// IOs for EL3446
	{attribute 'TcLinkTo' := 'TIID^Device 2 (EtherCAT)^Term 1 (EK1200)^Term 3 (EL3446)^I1 Channel^Overcurrent'}
	MDP5001_342_I1_Channel_Overcurrent_1						AT%I*  : BOOL;
	{attribute 'TcLinkTo' := 'TIID^Device 2 (EtherCAT)^Term 1 (EK1200)^Term 3 (EL3446)^I1 Channel^Inaccurate Current'}
	MDP5001_342_I1_Channel_Inaccurate_Current_1				AT%I*  : BOOL;
	{attribute 'TcLinkTo' := 'TIID^Device 2 (EtherCAT)^Term 1 (EK1200)^Term 3 (EL3446)^I1 Channel^Current Guard Warning'}
	MDP5001_342_I1_Channel_Current_Guard_Warning_1			AT%I*  : bool;
	{attribute 'TcLinkTo' := 'TIID^Device 2 (EtherCAT)^Term 1 (EK1200)^Term 3 (EL3446)^I1 Channel^Current Guard Error'}
	MDP5001_342_I1_Channel_Current_Guard_Error_1				AT%I*  : bool;
	{attribute 'TcLinkTo' := 'TIID^Device 2 (EtherCAT)^Term 1 (EK1200)^Term 3 (EL3446)^I1 Channel^Apparent Power Guard Warning'}
	MDP5001_342_I1_Channel_Apparent_Power_Guard_Warning_1		AT%I*  : bool;
	{attribute 'TcLinkTo' := 'TIID^Device 2 (EtherCAT)^Term 1 (EK1200)^Term 3 (EL3446)^I1 Channel^Apparent Power Guard Error'}
	MDP5001_342_I1_Channel_Apparent_Power_Guard_Error_1		AT%I*  : bool;
	{attribute 'TcLinkTo' := 'TIID^Device 2 (EtherCAT)^Term 1 (EK1200)^Term 3 (EL3446)^I1 Channel^Active Power Guard Warning'}
	MDP5001_342_I1_Channel_Active_Power_Guard_Warning_1		AT%I*  : bool;
	{attribute 'TcLinkTo' := 'TIID^Device 2 (EtherCAT)^Term 1 (EK1200)^Term 3 (EL3446)^I1 Channel^Active Power Guard Error'}
	MDP5001_342_I1_Channel_Active_Power_Guard_Error_1			AT%I*  : bool;
	{attribute 'TcLinkTo' := 'TIID^Device 2 (EtherCAT)^Term 1 (EK1200)^Term 3 (EL3446)^I1 Channel^Reactive Power Guard Warning'}
	MDP5001_342_I1_Channel_Reactive_Power_Guard_Warning_1		AT%I*  : bool;
	{attribute 'TcLinkTo' := 'TIID^Device 2 (EtherCAT)^Term 1 (EK1200)^Term 3 (EL3446)^I1 Channel^Reactive Power Guard Error'}
	MDP5001_342_I1_Channel_Reactive_Power_Guard_Error_1		AT%I*  : bool;
	{attribute 'TcLinkTo' := 'TIID^Device 2 (EtherCAT)^Term 1 (EK1200)^Term 3 (EL3446)^I1 Channel^DPM Inaccurate'}
	MDP5001_342_I1_Channel_DPM_Inaccurate_1					AT%I*  : bool;
	{attribute 'TcLinkTo' := 'TIID^Device 2 (EtherCAT)^Term 1 (EK1200)^Term 3 (EL3446)^I1 Channel^DPM Timeout'}
	MDP5001_342_I1_Channel_DPM_Timeout_1						AT%I*  : bool;
	{attribute 'TcLinkTo' := 'TIID^Device 2 (EtherCAT)^Term 1 (EK1200)^Term 3 (EL3446)^I1 Channel^TxPDO Toggle'}
	MDP5001_342_I1_Channel_TxPDO_Toggle_1						AT%I*  : bool;
	{attribute 'TcLinkTo' := 'TIID^Device 2 (EtherCAT)^Term 1 (EK1200)^Term 3 (EL3446)^I1 Channel^Current'}
	MDP5001_342_I1_Channel_Current_1							AT%I*  : REAL;
	{attribute 'TcLinkTo' := 'TIID^Device 2 (EtherCAT)^Term 1 (EK1200)^Term 3 (EL3446)^I1 Channel^Active Power'}
	MDP5001_342_I1_Channel_Active_Power_1						AT%I*  : REAL;
	{attribute 'TcLinkTo' := 'TIID^Device 2 (EtherCAT)^Term 1 (EK1200)^Term 3 (EL3446)^I1 Channel^Apparent Power'}
	MDP5001_342_I1_Channel_Apparent_Power_1					AT%I*  : REAL;
	{attribute 'TcLinkTo' := 'TIID^Device 2 (EtherCAT)^Term 1 (EK1200)^Term 3 (EL3446)^I1 Channel^Reactive Power Fundamental'}
	MDP5001_342_I1_Channel_Reactive_Power_Fundamental_1		AT%I*  : REAL;
	{attribute 'TcLinkTo' := 'TIID^Device 2 (EtherCAT)^Term 1 (EK1200)^Term 3 (EL3446)^I1 Channel^Active Energy'}
	MDP5001_342_I1_Channel_Active_Energy_1					AT%I*  : DINT;
	{attribute 'TcLinkTo' := 'TIID^Device 2 (EtherCAT)^Term 1 (EK1200)^Term 3 (EL3446)^I2 Channel^Overcurrent'}
	MDP5001_342_I2_Channel_Overcurrent_1						AT%I*  : BOOL;
	{attribute 'TcLinkTo' := 'TIID^Device 2 (EtherCAT)^Term 1 (EK1200)^Term 3 (EL3446)^I2 Channel^Inaccurate Current'}
	MDP5001_342_I2_Channel_Inaccurate_Current_1				AT%I*  : BOOL;
	{attribute 'TcLinkTo' := 'TIID^Device 2 (EtherCAT)^Term 1 (EK1200)^Term 3 (EL3446)^I2 Channel^Current Guard Warning'}
	MDP5001_342_I2_Channel_Current_Guard_Warning_1			AT%I*  : bool;
	{attribute 'TcLinkTo' := 'TIID^Device 2 (EtherCAT)^Term 1 (EK1200)^Term 3 (EL3446)^I2 Channel^Current Guard Error'}
	MDP5001_342_I2_Channel_Current_Guard_Error_1				AT%I*  : bool;
	{attribute 'TcLinkTo' := 'TIID^Device 2 (EtherCAT)^Term 1 (EK1200)^Term 3 (EL3446)^I2 Channel^Apparent Power Guard Warning'}
	MDP5001_342_I2_Channel_Apparent_Power_Guard_Warning_1		AT%I*  : bool;
	{attribute 'TcLinkTo' := 'TIID^Device 2 (EtherCAT)^Term 1 (EK1200)^Term 3 (EL3446)^I2 Channel^Apparent Power Guard Error'}
	MDP5001_342_I2_Channel_Apparent_Power_Guard_Error_1		AT%I*  : bool;
	{attribute 'TcLinkTo' := 'TIID^Device 2 (EtherCAT)^Term 1 (EK1200)^Term 3 (EL3446)^I2 Channel^Active Power Guard Warning'}
	MDP5001_342_I2_Channel_Active_Power_Guard_Warning_1		AT%I*  : bool;
	{attribute 'TcLinkTo' := 'TIID^Device 2 (EtherCAT)^Term 1 (EK1200)^Term 3 (EL3446)^I2 Channel^Active Power Guard Error'}
	MDP5001_342_I2_Channel_Active_Power_Guard_Error_1			AT%I*  : bool;
	{attribute 'TcLinkTo' := 'TIID^Device 2 (EtherCAT)^Term 1 (EK1200)^Term 3 (EL3446)^I2 Channel^Reactive Power Guard Warning'}
	MDP5001_342_I2_Channel_Reactive_Power_Guard_Warning_1		AT%I*  : bool;
	{attribute 'TcLinkTo' := 'TIID^Device 2 (EtherCAT)^Term 1 (EK1200)^Term 3 (EL3446)^I2 Channel^Reactive Power Guard Error'}
	MDP5001_342_I2_Channel_Reactive_Power_Guard_Error_1		AT%I*  : bool;
	{attribute 'TcLinkTo' := 'TIID^Device 2 (EtherCAT)^Term 1 (EK1200)^Term 3 (EL3446)^I2 Channel^DPM Inaccurate'}
	MDP5001_342_I2_Channel_DPM_Inaccurate_1					AT%I*  : bool;
	{attribute 'TcLinkTo' := 'TIID^Device 2 (EtherCAT)^Term 1 (EK1200)^Term 3 (EL3446)^I2 Channel^DPM Timeout'}
	MDP5001_342_I2_Channel_DPM_Timeout_1						AT%I*  : bool;
	{attribute 'TcLinkTo' := 'TIID^Device 2 (EtherCAT)^Term 1 (EK1200)^Term 3 (EL3446)^I2 Channel^TxPDO Toggle'}
	MDP5001_342_I2_Channel_TxPDO_Toggle_1						AT%I*  : bool;
	{attribute 'TcLinkTo' := 'TIID^Device 2 (EtherCAT)^Term 1 (EK1200)^Term 3 (EL3446)^I2 Channel^Current'}
	MDP5001_342_I2_Channel_Current_1							AT%I*  : REAL;
	{attribute 'TcLinkTo' := 'TIID^Device 2 (EtherCAT)^Term 1 (EK1200)^Term 3 (EL3446)^I2 Channel^Active Power'}
	MDP5001_342_I2_Channel_Active_Power_1						AT%I*  : REAL;
	{attribute 'TcLinkTo' := 'TIID^Device 2 (EtherCAT)^Term 1 (EK1200)^Term 3 (EL3446)^I2 Channel^Apparent Power'}
	MDP5001_342_I2_Channel_Apparent_Power_1					AT%I*  : REAL;
	{attribute 'TcLinkTo' := 'TIID^Device 2 (EtherCAT)^Term 1 (EK1200)^Term 3 (EL3446)^I2 Channel^Reactive Power Fundamental'}
	MDP5001_342_I2_Channel_Reactive_Power_Fundamental_1		AT%I*  : REAL;
	{attribute 'TcLinkTo' := 'TIID^Device 2 (EtherCAT)^Term 1 (EK1200)^Term 3 (EL3446)^I2 Channel^Active Energy'}
	MDP5001_342_I2_Channel_Active_Energy_1					AT%I*  : DINT;
	{attribute 'TcLinkTo' := 'TIID^Device 2 (EtherCAT)^Term 1 (EK1200)^Term 3 (EL3446)^I3 Channel^Overcurrent'}
	MDP5001_342_I3_Channel_Overcurrent_1						AT%I*  : BOOL;
	{attribute 'TcLinkTo' := 'TIID^Device 2 (EtherCAT)^Term 1 (EK1200)^Term 3 (EL3446)^I3 Channel^Inaccurate Current'}
	MDP5001_342_I3_Channel_Inaccurate_Current_1				AT%I*  : BOOL;
	{attribute 'TcLinkTo' := 'TIID^Device 2 (EtherCAT)^Term 1 (EK1200)^Term 3 (EL3446)^I3 Channel^Current Guard Warning'}
	MDP5001_342_I3_Channel_Current_Guard_Warning_1			AT%I*  : bool;
	{attribute 'TcLinkTo' := 'TIID^Device 2 (EtherCAT)^Term 1 (EK1200)^Term 3 (EL3446)^I3 Channel^Current Guard Error'}
	MDP5001_342_I3_Channel_Current_Guard_Error_1				AT%I*  : bool;
	{attribute 'TcLinkTo' := 'TIID^Device 2 (EtherCAT)^Term 1 (EK1200)^Term 3 (EL3446)^I3 Channel^Apparent Power Guard Warning'}
	MDP5001_342_I3_Channel_Apparent_Power_Guard_Warning_1		AT%I*  : bool;
	{attribute 'TcLinkTo' := 'TIID^Device 2 (EtherCAT)^Term 1 (EK1200)^Term 3 (EL3446)^I3 Channel^Apparent Power Guard Error'}
	MDP5001_342_I3_Channel_Apparent_Power_Guard_Error_1		AT%I*  : bool;
	{attribute 'TcLinkTo' := 'TIID^Device 2 (EtherCAT)^Term 1 (EK1200)^Term 3 (EL3446)^I3 Channel^Active Power Guard Warning'}
	MDP5001_342_I3_Channel_Active_Power_Guard_Warning_1		AT%I*  : bool;
	{attribute 'TcLinkTo' := 'TIID^Device 2 (EtherCAT)^Term 1 (EK1200)^Term 3 (EL3446)^I3 Channel^Active Power Guard Error'}
	MDP5001_342_I3_Channel_Active_Power_Guard_Error_1		AT%I*  : bool;
	{attribute 'TcLinkTo' := 'TIID^Device 2 (EtherCAT)^Term 1 (EK1200)^Term 3 (EL3446)^I3 Channel^Reactive Power Guard Warning'}
	MDP5001_342_I3_Channel_Reactive_Power_Guard_Warning_1		AT%I*  : bool;
	{attribute 'TcLinkTo' := 'TIID^Device 2 (EtherCAT)^Term 1 (EK1200)^Term 3 (EL3446)^I3 Channel^Reactive Power Guard Error'}
	MDP5001_342_I3_Channel_Reactive_Power_Guard_Error_1		AT%I*  : bool;
	{attribute 'TcLinkTo' := 'TIID^Device 2 (EtherCAT)^Term 1 (EK1200)^Term 3 (EL3446)^I3 Channel^DPM Inaccurate'}
	MDP5001_342_I3_Channel_DPM_Inaccurate_1					AT%I*  : bool;
	{attribute 'TcLinkTo' := 'TIID^Device 2 (EtherCAT)^Term 1 (EK1200)^Term 3 (EL3446)^I3 Channel^DPM Timeout'}
	MDP5001_342_I3_Channel_DPM_Timeout_1						AT%I*  : bool;
	{attribute 'TcLinkTo' := 'TIID^Device 2 (EtherCAT)^Term 1 (EK1200)^Term 3 (EL3446)^I3 Channel^TxPDO Toggle'}
	MDP5001_342_I3_Channel_TxPDO_Toggle_1						AT%I*  : bool;
	{attribute 'TcLinkTo' := 'TIID^Device 2 (EtherCAT)^Term 1 (EK1200)^Term 3 (EL3446)^I3 Channel^Current'}
	MDP5001_342_I3_Channel_Current_1							AT%I*  : REAL;
	{attribute 'TcLinkTo' := 'TIID^Device 2 (EtherCAT)^Term 1 (EK1200)^Term 3 (EL3446)^I3 Channel^Active Power'}
	MDP5001_342_I3_Channel_Active_Power_1						AT%I*  : REAL;
	{attribute 'TcLinkTo' := 'TIID^Device 2 (EtherCAT)^Term 1 (EK1200)^Term 3 (EL3446)^I3 Channel^Apparent Power'}
	MDP5001_342_I3_Channel_Apparent_Power_1					AT%I*  : REAL;
	{attribute 'TcLinkTo' := 'TIID^Device 2 (EtherCAT)^Term 1 (EK1200)^Term 3 (EL3446)^I3 Channel^Reactive Power Fundamental'}
	MDP5001_342_I3_Channel_Reactive_Power_Fundamental_1		AT%I*  : REAL;
	{attribute 'TcLinkTo' := 'TIID^Device 2 (EtherCAT)^Term 1 (EK1200)^Term 3 (EL3446)^I3 Channel^Active Energy'}
	MDP5001_342_I3_Channel_Active_Energy_1					AT%I*  : DINT;	
	{attribute 'TcLinkTo' := 'TIID^Device 2 (EtherCAT)^Term 1 (EK1200)^Term 3 (EL3446)^I4 Channel^Overcurrent'}
	MDP5001_342_I4_Channel_Overcurrent_1						AT%I*  : BOOL;
	{attribute 'TcLinkTo' := 'TIID^Device 2 (EtherCAT)^Term 1 (EK1200)^Term 3 (EL3446)^I4 Channel^Inaccurate Current'}
	MDP5001_342_I4_Channel_Inaccurate_Current_1				AT%I*  : BOOL;
	{attribute 'TcLinkTo' := 'TIID^Device 2 (EtherCAT)^Term 1 (EK1200)^Term 3 (EL3446)^I4 Channel^Current Guard Warning'}
	MDP5001_342_I4_Channel_Current_Guard_Warning_1			AT%I*  : bool;
	{attribute 'TcLinkTo' := 'TIID^Device 2 (EtherCAT)^Term 1 (EK1200)^Term 3 (EL3446)^I4 Channel^Current Guard Error'}
	MDP5001_342_I4_Channel_Current_Guard_Error_1				AT%I*  : bool;
	{attribute 'TcLinkTo' := 'TIID^Device 2 (EtherCAT)^Term 1 (EK1200)^Term 3 (EL3446)^I4 Channel^Apparent Power Guard Warning'}
	MDP5001_342_I4_Channel_Apparent_Power_Guard_Warning_1		AT%I*  : bool;
	{attribute 'TcLinkTo' := 'TIID^Device 2 (EtherCAT)^Term 1 (EK1200)^Term 3 (EL3446)^I4 Channel^Apparent Power Guard Error'}
	MDP5001_342_I4_Channel_Apparent_Power_Guard_Error_1		AT%I*  : bool;
	{attribute 'TcLinkTo' := 'TIID^Device 2 (EtherCAT)^Term 1 (EK1200)^Term 3 (EL3446)^I4 Channel^Active Power Guard Warning'}
	MDP5001_342_I4_Channel_Active_Power_Guard_Warning_1		AT%I*  : bool;
	{attribute 'TcLinkTo' := 'TIID^Device 2 (EtherCAT)^Term 1 (EK1200)^Term 3 (EL3446)^I4 Channel^Active Power Guard Error'}
	MDP5001_342_I4_Channel_Active_Power_Guard_Error_1			AT%I*  : bool;
	{attribute 'TcLinkTo' := 'TIID^Device 2 (EtherCAT)^Term 1 (EK1200)^Term 3 (EL3446)^I4 Channel^Reactive Power Guard Warning'}
	MDP5001_342_I4_Channel_Reactive_Power_Guard_Warning_1		AT%I*  : bool;
	{attribute 'TcLinkTo' := 'TIID^Device 2 (EtherCAT)^Term 1 (EK1200)^Term 3 (EL3446)^I4 Channel^Reactive Power Guard Error'}
	MDP5001_342_I4_Channel_Reactive_Power_Guard_Error_1		AT%I*  : bool;
	{attribute 'TcLinkTo' := 'TIID^Device 2 (EtherCAT)^Term 1 (EK1200)^Term 3 (EL3446)^I4 Channel^DPM Inaccurate'}
	MDP5001_342_I4_Channel_DPM_Inaccurate_1					AT%I*  : bool;
	{attribute 'TcLinkTo' := 'TIID^Device 2 (EtherCAT)^Term 1 (EK1200)^Term 3 (EL3446)^I4 Channel^DPM Timeout'}
	MDP5001_342_I4_Channel_DPM_Timeout_1						AT%I*  : bool;
	{attribute 'TcLinkTo' := 'TIID^Device 2 (EtherCAT)^Term 1 (EK1200)^Term 3 (EL3446)^I4 Channel^TxPDO Toggle'}
	MDP5001_342_I4_Channel_TxPDO_Toggle_1						AT%I*  : bool;
	{attribute 'TcLinkTo' := 'TIID^Device 2 (EtherCAT)^Term 1 (EK1200)^Term 3 (EL3446)^I4 Channel^Current'}
	MDP5001_342_I4_Channel_Current_1							AT%I*  : REAL;
	{attribute 'TcLinkTo' := 'TIID^Device 2 (EtherCAT)^Term 1 (EK1200)^Term 3 (EL3446)^I4 Channel^Active Power'}
	MDP5001_342_I4_Channel_Active_Power_1						AT%I*  : REAL;
	{attribute 'TcLinkTo' := 'TIID^Device 2 (EtherCAT)^Term 1 (EK1200)^Term 3 (EL3446)^I4 Channel^Apparent Power'}
	MDP5001_342_I4_Channel_Apparent_Power_1					AT%I*  : REAL;
	{attribute 'TcLinkTo' := 'TIID^Device 2 (EtherCAT)^Term 1 (EK1200)^Term 3 (EL3446)^I4 Channel^Reactive Power Fundamental'}
	MDP5001_342_I4_Channel_Reactive_Power_Fundamental_1		AT%I*  : REAL;
	{attribute 'TcLinkTo' := 'TIID^Device 2 (EtherCAT)^Term 1 (EK1200)^Term 3 (EL3446)^I4 Channel^Active Energy'}
	MDP5001_342_I4_Channel_Active_Energy_1					AT%I*  : DINT;
	{attribute 'TcLinkTo' := 'TIID^Device 2 (EtherCAT)^Term 1 (EK1200)^Term 3 (EL3446)^I5 Channel^Overcurrent'}
	MDP5001_342_I5_Channel_Overcurrent_1						AT%I*  : BOOL;
	{attribute 'TcLinkTo' := 'TIID^Device 2 (EtherCAT)^Term 1 (EK1200)^Term 3 (EL3446)^I5 Channel^Inaccurate Current'}
	MDP5001_342_I5_Channel_Inaccurate_Current_1				AT%I*  : BOOL;
	{attribute 'TcLinkTo' := 'TIID^Device 2 (EtherCAT)^Term 1 (EK1200)^Term 3 (EL3446)^I5 Channel^Current Guard Warning'}
	MDP5001_342_I5_Channel_Current_Guard_Warning_1			AT%I*  : bool;
	{attribute 'TcLinkTo' := 'TIID^Device 2 (EtherCAT)^Term 1 (EK1200)^Term 3 (EL3446)^I5 Channel^Current Guard Error'}
	MDP5001_342_I5_Channel_Current_Guard_Error_1				AT%I*  : bool;
	{attribute 'TcLinkTo' := 'TIID^Device 2 (EtherCAT)^Term 1 (EK1200)^Term 3 (EL3446)^I5 Channel^Apparent Power Guard Warning'}
	MDP5001_342_I5_Channel_Apparent_Power_Guard_Warning_1		AT%I*  : bool;
	{attribute 'TcLinkTo' := 'TIID^Device 2 (EtherCAT)^Term 1 (EK1200)^Term 3 (EL3446)^I5 Channel^Apparent Power Guard Error'}
	MDP5001_342_I5_Channel_Apparent_Power_Guard_Error_1		AT%I*  : bool;
	{attribute 'TcLinkTo' := 'TIID^Device 2 (EtherCAT)^Term 1 (EK1200)^Term 3 (EL3446)^I5 Channel^Active Power Guard Warning'}
	MDP5001_342_I5_Channel_Active_Power_Guard_Warning_1		AT%I*  : bool;
	{attribute 'TcLinkTo' := 'TIID^Device 2 (EtherCAT)^Term 1 (EK1200)^Term 3 (EL3446)^I5 Channel^Active Power Guard Error'}
	MDP5001_342_I5_Channel_Active_Power_Guard_Error_1			AT%I*  : bool;
	{attribute 'TcLinkTo' := 'TIID^Device 2 (EtherCAT)^Term 1 (EK1200)^Term 3 (EL3446)^I5 Channel^Reactive Power Guard Warning'}
	MDP5001_342_I5_Channel_Reactive_Power_Guard_Warning_1		AT%I*  : bool;
	{attribute 'TcLinkTo' := 'TIID^Device 2 (EtherCAT)^Term 1 (EK1200)^Term 3 (EL3446)^I5 Channel^Reactive Power Guard Error'}
	MDP5001_342_I5_Channel_Reactive_Power_Guard_Error_1		AT%I*  : bool;
	{attribute 'TcLinkTo' := 'TIID^Device 2 (EtherCAT)^Term 1 (EK1200)^Term 3 (EL3446)^I5 Channel^DPM Inaccurate'}
	MDP5001_342_I5_Channel_DPM_Inaccurate_1					AT%I*  : bool;
	{attribute 'TcLinkTo' := 'TIID^Device 2 (EtherCAT)^Term 1 (EK1200)^Term 3 (EL3446)^I5 Channel^DPM Timeout'}
	MDP5001_342_I5_Channel_DPM_Timeout_1						AT%I*  : bool;
	{attribute 'TcLinkTo' := 'TIID^Device 2 (EtherCAT)^Term 1 (EK1200)^Term 3 (EL3446)^I5 Channel^TxPDO Toggle'}
	MDP5001_342_I5_Channel_TxPDO_Toggle_1						AT%I*  : bool;
	{attribute 'TcLinkTo' := 'TIID^Device 2 (EtherCAT)^Term 1 (EK1200)^Term 3 (EL3446)^I5 Channel^Current'}
	MDP5001_342_I5_Channel_Current_1							AT%I*  : REAL;
	{attribute 'TcLinkTo' := 'TIID^Device 2 (EtherCAT)^Term 1 (EK1200)^Term 3 (EL3446)^I5 Channel^Active Power'}
	MDP5001_342_I5_Channel_Active_Power_1						AT%I*  : REAL;
	{attribute 'TcLinkTo' := 'TIID^Device 2 (EtherCAT)^Term 1 (EK1200)^Term 3 (EL3446)^I5 Channel^Apparent Power'}
	MDP5001_342_I5_Channel_Apparent_Power_1					AT%I*  : REAL;
	{attribute 'TcLinkTo' := 'TIID^Device 2 (EtherCAT)^Term 1 (EK1200)^Term 3 (EL3446)^I5 Channel^Reactive Power Fundamental'}
	MDP5001_342_I5_Channel_Reactive_Power_Fundamental_1		AT%I*  : REAL;
	{attribute 'TcLinkTo' := 'TIID^Device 2 (EtherCAT)^Term 1 (EK1200)^Term 3 (EL3446)^I5 Channel^Active Energy'}
	MDP5001_342_I5_Channel_Active_Energy_1					AT%I*  : DINT;
	{attribute 'TcLinkTo' := 'TIID^Device 2 (EtherCAT)^Term 1 (EK1200)^Term 3 (EL3446)^I6 Channel^Overcurrent'}
	MDP5001_342_I6_Channel_Overcurrent_1						AT%I*  : BOOL;
	{attribute 'TcLinkTo' := 'TIID^Device 2 (EtherCAT)^Term 1 (EK1200)^Term 3 (EL3446)^I6 Channel^Inaccurate Current'}
	MDP5001_342_I6_Channel_Inaccurate_Current_1				AT%I*  : BOOL;
	{attribute 'TcLinkTo' := 'TIID^Device 2 (EtherCAT)^Term 1 (EK1200)^Term 3 (EL3446)^I6 Channel^Current Guard Warning'}
	MDP5001_342_I6_Channel_Current_Guard_Warning_1			AT%I*  : bool;
	{attribute 'TcLinkTo' := 'TIID^Device 2 (EtherCAT)^Term 1 (EK1200)^Term 3 (EL3446)^I6 Channel^Current Guard Error'}
	MDP5001_342_I6_Channel_Current_Guard_Error_1				AT%I*  : bool;
	{attribute 'TcLinkTo' := 'TIID^Device 2 (EtherCAT)^Term 1 (EK1200)^Term 3 (EL3446)^I6 Channel^Apparent Power Guard Warning'}
	MDP5001_342_I6_Channel_Apparent_Power_Guard_Warning_1		AT%I*  : bool;
	{attribute 'TcLinkTo' := 'TIID^Device 2 (EtherCAT)^Term 1 (EK1200)^Term 3 (EL3446)^I6 Channel^Apparent Power Guard Error'}
	MDP5001_342_I6_Channel_Apparent_Power_Guard_Error_1		AT%I*  : bool;
	{attribute 'TcLinkTo' := 'TIID^Device 2 (EtherCAT)^Term 1 (EK1200)^Term 3 (EL3446)^I6 Channel^Active Power Guard Warning'}
	MDP5001_342_I6_Channel_Active_Power_Guard_Warning_1		AT%I*  : bool;
	{attribute 'TcLinkTo' := 'TIID^Device 2 (EtherCAT)^Term 1 (EK1200)^Term 3 (EL3446)^I6 Channel^Active Power Guard Error'}
	MDP5001_342_I6_Channel_Active_Power_Guard_Error_1			AT%I*  : bool;
	{attribute 'TcLinkTo' := 'TIID^Device 2 (EtherCAT)^Term 1 (EK1200)^Term 3 (EL3446)^I6 Channel^Reactive Power Guard Warning'}
	MDP5001_342_I6_Channel_Reactive_Power_Guard_Warning_1		AT%I*  : bool;
	{attribute 'TcLinkTo' := 'TIID^Device 2 (EtherCAT)^Term 1 (EK1200)^Term 3 (EL3446)^I6 Channel^Reactive Power Guard Error'}
	MDP5001_342_I6_Channel_Reactive_Power_Guard_Error_1		AT%I*  : bool;
	{attribute 'TcLinkTo' := 'TIID^Device 2 (EtherCAT)^Term 1 (EK1200)^Term 3 (EL3446)^I6 Channel^DPM Inaccurate'}
	MDP5001_342_I6_Channel_DPM_Inaccurate_1					AT%I*  : bool;
	{attribute 'TcLinkTo' := 'TIID^Device 2 (EtherCAT)^Term 1 (EK1200)^Term 3 (EL3446)^I6 Channel^DPM Timeout'}
	MDP5001_342_I6_Channel_DPM_Timeout_1						AT%I*  : bool;
	{attribute 'TcLinkTo' := 'TIID^Device 2 (EtherCAT)^Term 1 (EK1200)^Term 3 (EL3446)^I6 Channel^TxPDO Toggle'}
	MDP5001_342_I6_Channel_TxPDO_Toggle_1						AT%I*  : bool;
	{attribute 'TcLinkTo' := 'TIID^Device 2 (EtherCAT)^Term 1 (EK1200)^Term 3 (EL3446)^I6 Channel^Current'}
	MDP5001_342_I6_Channel_Current_1							AT%I*  : REAL;
	{attribute 'TcLinkTo' := 'TIID^Device 2 (EtherCAT)^Term 1 (EK1200)^Term 3 (EL3446)^I6 Channel^Active Power'}
	MDP5001_342_I6_Channel_Active_Power_1						AT%I*  : REAL;
	{attribute 'TcLinkTo' := 'TIID^Device 2 (EtherCAT)^Term 1 (EK1200)^Term 3 (EL3446)^I6 Channel^Apparent Power'}
	MDP5001_342_I6_Channel_Apparent_Power_1					AT%I*  : REAL;
	{attribute 'TcLinkTo' := 'TIID^Device 2 (EtherCAT)^Term 1 (EK1200)^Term 3 (EL3446)^I6 Channel^Reactive Power Fundamental'}
	MDP5001_342_I6_Channel_Reactive_Power_Fundamental_1		AT%I*  : REAL;
	{attribute 'TcLinkTo' := 'TIID^Device 2 (EtherCAT)^Term 1 (EK1200)^Term 3 (EL3446)^I6 Channel^Active Energy'}
	MDP5001_342_I6_Channel_Active_Energy_1					AT%I*  : DINT;	
	
	{attribute 'TcLinkTo' := 'TIID^Device 2 (EtherCAT)^Term 1 (EK1200)^Term 3 (EL3446)^DPM Variant Value In^TxPDO Toggle'}
	MDP5001_342_DPM_Variant_Value_In_TxPDO_Toggle_1			AT%I*  : BOOL;
	{attribute 'TcLinkTo' := 'TIID^Device 2 (EtherCAT)^Term 1 (EK1200)^Term 3 (EL3446)^DPM Variant Value In^Index 1 REAL'}
	MDP5001_342_DPM_Variant_Value_In_Index_1_REAL_1			AT%I*  : UINT;
	{attribute 'TcLinkTo' := 'TIID^Device 2 (EtherCAT)^Term 1 (EK1200)^Term 3 (EL3446)^DPM Variant Value In^Value 1 REAL'}
	MDP5001_342_DPM_Variant_Value_In_Value_1_REAL_1			AT%I*  : REAL;
	{attribute 'TcLinkTo' := 'TIID^Device 2 (EtherCAT)^Term 1 (EK1200)^Term 3 (EL3446)^DPM Variant Value In^Index 2 REAL'}
	MDP5001_342_DPM_Variant_Value_In_Index_2_REAL_1			AT%I*  : UINT;
	{attribute 'TcLinkTo' := 'TIID^Device 2 (EtherCAT)^Term 1 (EK1200)^Term 3 (EL3446)^DPM Variant Value In^Value 2 REAL'}
	MDP5001_342_DPM_Variant_Value_In_Value_2_REAL_1			AT%I*  : REAL;
	{attribute 'TcLinkTo' := 'TIID^Device 2 (EtherCAT)^Term 1 (EK1200)^Term 3 (EL3446)^DPM Variant Value In^Index 3 REAL'}
	MDP5001_342_DPM_Variant_Value_In_Index_3_REAL_1			AT%I*  : UINT;
	{attribute 'TcLinkTo' := 'TIID^Device 2 (EtherCAT)^Term 1 (EK1200)^Term 3 (EL3446)^DPM Variant Value In^Value 3 REAL'}
	MDP5001_342_DPM_Variant_Value_In_Value_3_REAL_1			AT%I*  : REAL;
	{attribute 'TcLinkTo' := 'TIID^Device 2 (EtherCAT)^Term 1 (EK1200)^Term 3 (EL3446)^DPM Variant Value In^Index 4 ULINT'}
	MDP5001_342_DPM_Variant_Value_In_Index_4_ULINT_1			AT%I*  : UINT;
	{attribute 'TcLinkTo' := 'TIID^Device 2 (EtherCAT)^Term 1 (EK1200)^Term 3 (EL3446)^DPM Variant Value In^Value 4 ULINT'}
	MDP5001_342_DPM_Variant_Value_In_Value_4_ULINT_1			AT%I*  : ULINT;

	{attribute 'TcLinkTo' := 'TIID^Device 2 (EtherCAT)^Term 1 (EK1200)^Term 3 (EL3446)^DPM Variant Value Out^Index 1 REAL'}
	MDP5001_342_DPM_Variant_Value_Out_Index_1_REAL_1	AT%Q* : UINT;
	{attribute 'TcLinkTo' := 'TIID^Device 2 (EtherCAT)^Term 1 (EK1200)^Term 3 (EL3446)^DPM Variant Value Out^Index 2 REAL'}
	MDP5001_342_DPM_Variant_Value_Out_Index_2_REAL_1	AT%Q* : UINT;
	{attribute 'TcLinkTo' := 'TIID^Device 2 (EtherCAT)^Term 1 (EK1200)^Term 3 (EL3446)^DPM Variant Value Out^Index 3 REAL'}
	MDP5001_342_DPM_Variant_Value_Out_Index_3_REAL_1	AT%Q* : UINT;
	{attribute 'TcLinkTo' := 'TIID^Device 2 (EtherCAT)^Term 1 (EK1200)^Term 3 (EL3446)^DPM Variant Value Out^Index 4 ULINT'}
	MDP5001_342_DPM_Variant_Value_Out_Index_4_ULINT_1	AT%Q* : UINT;
	{attribute 'TcLinkTo' := 'TIID^Device 2 (EtherCAT)^Term 1 (EK1200)^Term 3 (EL3446)^DPM Data^Data 1'}
	MDP5001_342_DPM_Data_Data_1_1						AT%Q* : UDINT;
	{attribute 'TcLinkTo' := 'TIID^Device 2 (EtherCAT)^Term 1 (EK1200)^Term 3 (EL3446)^DPM Data^Data 2'}
	MDP5001_342_DPM_Data_Data_2_1						AT%Q* : UDINT;
	{attribute 'TcLinkTo' := 'TIID^Device 2 (EtherCAT)^Term 1 (EK1200)^Term 3 (EL3446)^DPM Data^Data 3'}
	MDP5001_342_DPM_Data_Data_3_1						AT%Q* : UDINT;
	{attribute 'TcLinkTo' := 'TIID^Device 2 (EtherCAT)^Term 1 (EK1200)^Term 3 (EL3446)^DPM Data^Data 4'}
	MDP5001_342_DPM_Data_Data_4_1						AT%Q* : UDINT;
	{attribute 'TcLinkTo' := 'TIID^Device 2 (EtherCAT)^Term 1 (EK1200)^Term 3 (EL3446)^DPM Data^Data 5'}
	MDP5001_342_DPM_Data_Data_5_1						AT%Q* : UDINT;
	{attribute 'TcLinkTo' := 'TIID^Device 2 (EtherCAT)^Term 1 (EK1200)^Term 3 (EL3446)^DPM Data^Data 6'}
	MDP5001_342_DPM_Data_Data_6_1						AT%Q* : UDINT;
	{attribute 'TcLinkTo' := 'TIID^Device 2 (EtherCAT)^Term 1 (EK1200)^Term 3 (EL3446)^DPM Data^Data 7'}
	MDP5001_342_DPM_Data_Data_7_1						AT%Q* : UDINT;
	{attribute 'TcLinkTo' := 'TIID^Device 2 (EtherCAT)^Term 1 (EK1200)^Term 3 (EL3446)^DPM Data^Data 8'}
	MDP5001_342_DPM_Data_Data_8_1						AT%Q* : UDINT;
	{attribute 'TcLinkTo' := 'TIID^Device 2 (EtherCAT)^Term 1 (EK1200)^Term 3 (EL3446)^DPM Data^Data 9'}
	MDP5001_342_DPM_Data_Data_9_1						AT%Q* : UDINT;
	{attribute 'TcLinkTo' := 'TIID^Device 2 (EtherCAT)^Term 1 (EK1200)^Term 3 (EL3446)^DPM Data^Data 10'}
	MDP5001_342_DPM_Data_Data_10_1					AT%Q* : UDINT;
	{attribute 'TcLinkTo' := 'TIID^Device 2 (EtherCAT)^Term 1 (EK1200)^Term 3 (EL3446)^DPM Data^Data 11'}
	MDP5001_342_DPM_Data_Data_11_1					AT%Q* : UDINT;
	{attribute 'TcLinkTo' := 'TIID^Device 2 (EtherCAT)^Term 1 (EK1200)^Term 3 (EL3446)^DPM Data^Data 12'}
	MDP5001_342_DPM_Data_Data_12_1					AT%Q* : UDINT;
	{attribute 'TcLinkTo' := 'TIID^Device 2 (EtherCAT)^Term 1 (EK1200)^Term 3 (EL3446)^DPM Data^Data 13'}
	MDP5001_342_DPM_Data_Data_13_1					AT%Q* : UDINT;
	{attribute 'TcLinkTo' := 'TIID^Device 2 (EtherCAT)^Term 1 (EK1200)^Term 3 (EL3446)^DPM Data^Data 14'}
	MDP5001_342_DPM_Data_Data_14_1					AT%Q* : UDINT;
	{attribute 'TcLinkTo' := 'TIID^Device 2 (EtherCAT)^Term 1 (EK1200)^Term 3 (EL3446)^DPM Data^Data 15'}
	MDP5001_342_DPM_Data_Data_15_1					AT%Q* : UDINT;
	{attribute 'TcLinkTo' := 'TIID^Device 2 (EtherCAT)^Term 1 (EK1200)^Term 3 (EL3446)^DPM Data^Data 16'}
	MDP5001_342_DPM_Data_Data_16_1					AT%Q* : UDINT;
	{attribute 'TcLinkTo' := 'TIID^Device 2 (EtherCAT)^Term 1 (EK1200)^Term 3 (EL3446)^DPM Data^Data 17'}
	MDP5001_342_DPM_Data_Data_17_1					AT%Q* : UDINT;
	{attribute 'TcLinkTo' := 'TIID^Device 2 (EtherCAT)^Term 1 (EK1200)^Term 3 (EL3446)^DPM Data^Data 18'}
	MDP5001_342_DPM_Data_Data_18_1					AT%Q* : UDINT;
	{attribute 'TcLinkTo' := 'TIID^Device 2 (EtherCAT)^Term 1 (EK1200)^Term 3 (EL3446)^DPM Data^Data 19'}
	MDP5001_342_DPM_Data_Data_19_1					AT%Q* : UDINT;
	{attribute 'TcLinkTo' := 'TIID^Device 2 (EtherCAT)^Term 1 (EK1200)^Term 3 (EL3446)^DPM Data^Data 20'}
	MDP5001_342_DPM_Data_Data_20_1					AT%Q* : UDINT;



// IOs for EL3446
	{attribute 'TcLinkTo' := 'TIID^Device 2 (EtherCAT)^Term 1 (EK1200)^Term 4 (EL3446)^I1 Channel^Overcurrent'}
	MDP5001_342_I1_Channel_Overcurrent_2						AT%I*  : BOOL;
	{attribute 'TcLinkTo' := 'TIID^Device 2 (EtherCAT)^Term 1 (EK1200)^Term 4 (EL3446)^I1 Channel^Inaccurate Current'}
	MDP5001_342_I1_Channel_Inaccurate_Current_2				AT%I*  : BOOL;
	{attribute 'TcLinkTo' := 'TIID^Device 2 (EtherCAT)^Term 1 (EK1200)^Term 4 (EL3446)^I1 Channel^Current Guard Warning'}
	MDP5001_342_I1_Channel_Current_Guard_Warning_2			AT%I*  : bool;
	{attribute 'TcLinkTo' := 'TIID^Device 2 (EtherCAT)^Term 1 (EK1200)^Term 4 (EL3446)^I1 Channel^Current Guard Error'}
	MDP5001_342_I1_Channel_Current_Guard_Error_2				AT%I*  : bool;
	{attribute 'TcLinkTo' := 'TIID^Device 2 (EtherCAT)^Term 1 (EK1200)^Term 4 (EL3446)^I1 Channel^Apparent Power Guard Warning'}
	MDP5001_342_I1_Channel_Apparent_Power_Guard_Warning_2		AT%I*  : bool;
	{attribute 'TcLinkTo' := 'TIID^Device 2 (EtherCAT)^Term 1 (EK1200)^Term 4 (EL3446)^I1 Channel^Apparent Power Guard Error'}
	MDP5001_342_I1_Channel_Apparent_Power_Guard_Error_2		AT%I*  : bool;
	{attribute 'TcLinkTo' := 'TIID^Device 2 (EtherCAT)^Term 1 (EK1200)^Term 4 (EL3446)^I1 Channel^Active Power Guard Warning'}
	MDP5001_342_I1_Channel_Active_Power_Guard_Warning_2		AT%I*  : bool;
	{attribute 'TcLinkTo' := 'TIID^Device 2 (EtherCAT)^Term 1 (EK1200)^Term 4 (EL3446)^I1 Channel^Active Power Guard Error'}
	MDP5001_342_I1_Channel_Active_Power_Guard_Error_2			AT%I*  : bool;
	{attribute 'TcLinkTo' := 'TIID^Device 2 (EtherCAT)^Term 1 (EK1200)^Term 4 (EL3446)^I1 Channel^Reactive Power Guard Warning'}
	MDP5001_342_I1_Channel_Reactive_Power_Guard_Warning_2		AT%I*  : bool;
	{attribute 'TcLinkTo' := 'TIID^Device 2 (EtherCAT)^Term 1 (EK1200)^Term 4 (EL3446)^I1 Channel^Reactive Power Guard Error'}
	MDP5001_342_I1_Channel_Reactive_Power_Guard_Error_2		AT%I*  : bool;
	{attribute 'TcLinkTo' := 'TIID^Device 2 (EtherCAT)^Term 1 (EK1200)^Term 4 (EL3446)^I1 Channel^DPM Inaccurate'}
	MDP5001_342_I1_Channel_DPM_Inaccurate_2					AT%I*  : bool;
	{attribute 'TcLinkTo' := 'TIID^Device 2 (EtherCAT)^Term 1 (EK1200)^Term 4 (EL3446)^I1 Channel^DPM Timeout'}
	MDP5001_342_I1_Channel_DPM_Timeout_2						AT%I*  : bool;
	{attribute 'TcLinkTo' := 'TIID^Device 2 (EtherCAT)^Term 1 (EK1200)^Term 4 (EL3446)^I1 Channel^TxPDO Toggle'}
	MDP5001_342_I1_Channel_TxPDO_Toggle_2						AT%I*  : bool;
	{attribute 'TcLinkTo' := 'TIID^Device 2 (EtherCAT)^Term 1 (EK1200)^Term 4 (EL3446)^I1 Channel^Current'}
	MDP5001_342_I1_Channel_Current_2							AT%I*  : REAL;
	{attribute 'TcLinkTo' := 'TIID^Device 2 (EtherCAT)^Term 1 (EK1200)^Term 4 (EL3446)^I1 Channel^Active Power'}
	MDP5001_342_I1_Channel_Active_Power_2						AT%I*  : REAL;
	{attribute 'TcLinkTo' := 'TIID^Device 2 (EtherCAT)^Term 1 (EK1200)^Term 4 (EL3446)^I1 Channel^Apparent Power'}
	MDP5001_342_I1_Channel_Apparent_Power_2					AT%I*  : REAL;
	{attribute 'TcLinkTo' := 'TIID^Device 2 (EtherCAT)^Term 1 (EK1200)^Term 4 (EL3446)^I1 Channel^Reactive Power Fundamental'}
	MDP5001_342_I1_Channel_Reactive_Power_Fundamental_2		AT%I*  : REAL;
	{attribute 'TcLinkTo' := 'TIID^Device 2 (EtherCAT)^Term 1 (EK1200)^Term 4 (EL3446)^I1 Channel^Active Energy'}
	MDP5001_342_I1_Channel_Active_Energy_2					AT%I*  : DINT;
	{attribute 'TcLinkTo' := 'TIID^Device 2 (EtherCAT)^Term 1 (EK1200)^Term 4 (EL3446)^I2 Channel^Overcurrent'}
	MDP5001_342_I2_Channel_Overcurrent_2						AT%I*  : BOOL;
	{attribute 'TcLinkTo' := 'TIID^Device 2 (EtherCAT)^Term 1 (EK1200)^Term 4 (EL3446)^I2 Channel^Inaccurate Current'}
	MDP5001_342_I2_Channel_Inaccurate_Current_2				AT%I*  : BOOL;
	{attribute 'TcLinkTo' := 'TIID^Device 2 (EtherCAT)^Term 1 (EK1200)^Term 4 (EL3446)^I2 Channel^Current Guard Warning'}
	MDP5001_342_I2_Channel_Current_Guard_Warning_2			AT%I*  : bool;
	{attribute 'TcLinkTo' := 'TIID^Device 2 (EtherCAT)^Term 1 (EK1200)^Term 4 (EL3446)^I2 Channel^Current Guard Error'}
	MDP5001_342_I2_Channel_Current_Guard_Error_2				AT%I*  : bool;
	{attribute 'TcLinkTo' := 'TIID^Device 2 (EtherCAT)^Term 1 (EK1200)^Term 4 (EL3446)^I2 Channel^Apparent Power Guard Warning'}
	MDP5001_342_I2_Channel_Apparent_Power_Guard_Warning_2		AT%I*  : bool;
	{attribute 'TcLinkTo' := 'TIID^Device 2 (EtherCAT)^Term 1 (EK1200)^Term 4 (EL3446)^I2 Channel^Apparent Power Guard Error'}
	MDP5001_342_I2_Channel_Apparent_Power_Guard_Error_2		AT%I*  : bool;
	{attribute 'TcLinkTo' := 'TIID^Device 2 (EtherCAT)^Term 1 (EK1200)^Term 4 (EL3446)^I2 Channel^Active Power Guard Warning'}
	MDP5001_342_I2_Channel_Active_Power_Guard_Warning_2		AT%I*  : bool;
	{attribute 'TcLinkTo' := 'TIID^Device 2 (EtherCAT)^Term 1 (EK1200)^Term 4 (EL3446)^I2 Channel^Active Power Guard Error'}
	MDP5001_342_I2_Channel_Active_Power_Guard_Error_2			AT%I*  : bool;
	{attribute 'TcLinkTo' := 'TIID^Device 2 (EtherCAT)^Term 1 (EK1200)^Term 4 (EL3446)^I2 Channel^Reactive Power Guard Warning'}
	MDP5001_342_I2_Channel_Reactive_Power_Guard_Warning_2		AT%I*  : bool;
	{attribute 'TcLinkTo' := 'TIID^Device 2 (EtherCAT)^Term 1 (EK1200)^Term 4 (EL3446)^I2 Channel^Reactive Power Guard Error'}
	MDP5001_342_I2_Channel_Reactive_Power_Guard_Error_2		AT%I*  : bool;
	{attribute 'TcLinkTo' := 'TIID^Device 2 (EtherCAT)^Term 1 (EK1200)^Term 4 (EL3446)^I2 Channel^DPM Inaccurate'}
	MDP5001_342_I2_Channel_DPM_Inaccurate_2					AT%I*  : bool;
	{attribute 'TcLinkTo' := 'TIID^Device 2 (EtherCAT)^Term 1 (EK1200)^Term 4 (EL3446)^I2 Channel^DPM Timeout'}
	MDP5001_342_I2_Channel_DPM_Timeout_2						AT%I*  : bool;
	{attribute 'TcLinkTo' := 'TIID^Device 2 (EtherCAT)^Term 1 (EK1200)^Term 4 (EL3446)^I2 Channel^TxPDO Toggle'}
	MDP5001_342_I2_Channel_TxPDO_Toggle_2						AT%I*  : bool;
	{attribute 'TcLinkTo' := 'TIID^Device 2 (EtherCAT)^Term 1 (EK1200)^Term 4 (EL3446)^I2 Channel^Current'}
	MDP5001_342_I2_Channel_Current_2							AT%I*  : REAL;
	{attribute 'TcLinkTo' := 'TIID^Device 2 (EtherCAT)^Term 1 (EK1200)^Term 4 (EL3446)^I2 Channel^Active Power'}
	MDP5001_342_I2_Channel_Active_Power_2						AT%I*  : REAL;
	{attribute 'TcLinkTo' := 'TIID^Device 2 (EtherCAT)^Term 1 (EK1200)^Term 4 (EL3446)^I2 Channel^Apparent Power'}
	MDP5001_342_I2_Channel_Apparent_Power_2					AT%I*  : REAL;
	{attribute 'TcLinkTo' := 'TIID^Device 2 (EtherCAT)^Term 1 (EK1200)^Term 4 (EL3446)^I2 Channel^Reactive Power Fundamental'}
	MDP5001_342_I2_Channel_Reactive_Power_Fundamental_2		AT%I*  : REAL;
	{attribute 'TcLinkTo' := 'TIID^Device 2 (EtherCAT)^Term 1 (EK1200)^Term 4 (EL3446)^I2 Channel^Active Energy'}
	MDP5001_342_I2_Channel_Active_Energy_2					AT%I*  : DINT;
	{attribute 'TcLinkTo' := 'TIID^Device 2 (EtherCAT)^Term 1 (EK1200)^Term 4 (EL3446)^I3 Channel^Overcurrent'}
	MDP5001_342_I3_Channel_Overcurrent_2						AT%I*  : BOOL;
	{attribute 'TcLinkTo' := 'TIID^Device 2 (EtherCAT)^Term 1 (EK1200)^Term 4 (EL3446)^I3 Channel^Inaccurate Current'}
	MDP5001_342_I3_Channel_Inaccurate_Current_2				AT%I*  : BOOL;
	{attribute 'TcLinkTo' := 'TIID^Device 2 (EtherCAT)^Term 1 (EK1200)^Term 4 (EL3446)^I3 Channel^Current Guard Warning'}
	MDP5001_342_I3_Channel_Current_Guard_Warning_2			AT%I*  : bool;
	{attribute 'TcLinkTo' := 'TIID^Device 2 (EtherCAT)^Term 1 (EK1200)^Term 4 (EL3446)^I3 Channel^Current Guard Error'}
	MDP5001_342_I3_Channel_Current_Guard_Error_2				AT%I*  : bool;
	{attribute 'TcLinkTo' := 'TIID^Device 2 (EtherCAT)^Term 1 (EK1200)^Term 4 (EL3446)^I3 Channel^Apparent Power Guard Warning'}
	MDP5001_342_I3_Channel_Apparent_Power_Guard_Warning_2		AT%I*  : bool;
	{attribute 'TcLinkTo' := 'TIID^Device 2 (EtherCAT)^Term 1 (EK1200)^Term 4 (EL3446)^I3 Channel^Apparent Power Guard Error'}
	MDP5001_342_I3_Channel_Apparent_Power_Guard_Error_2		AT%I*  : bool;
	{attribute 'TcLinkTo' := 'TIID^Device 2 (EtherCAT)^Term 1 (EK1200)^Term 4 (EL3446)^I3 Channel^Active Power Guard Warning'}
	MDP5001_342_I3_Channel_Active_Power_Guard_Warning_2		AT%I*  : bool;
	{attribute 'TcLinkTo' := 'TIID^Device 2 (EtherCAT)^Term 1 (EK1200)^Term 4 (EL3446)^I3 Channel^Active Power Guard Error'}
	MDP5001_342_I3_Channel_Active_Power_Guard_Error_2		AT%I*  : bool;
	{attribute 'TcLinkTo' := 'TIID^Device 2 (EtherCAT)^Term 1 (EK1200)^Term 4 (EL3446)^I3 Channel^Reactive Power Guard Warning'}
	MDP5001_342_I3_Channel_Reactive_Power_Guard_Warning_2		AT%I*  : bool;
	{attribute 'TcLinkTo' := 'TIID^Device 2 (EtherCAT)^Term 1 (EK1200)^Term 4 (EL3446)^I3 Channel^Reactive Power Guard Error'}
	MDP5001_342_I3_Channel_Reactive_Power_Guard_Error_2		AT%I*  : bool;
	{attribute 'TcLinkTo' := 'TIID^Device 2 (EtherCAT)^Term 1 (EK1200)^Term 4 (EL3446)^I3 Channel^DPM Inaccurate'}
	MDP5001_342_I3_Channel_DPM_Inaccurate_2					AT%I*  : bool;
	{attribute 'TcLinkTo' := 'TIID^Device 2 (EtherCAT)^Term 1 (EK1200)^Term 4 (EL3446)^I3 Channel^DPM Timeout'}
	MDP5001_342_I3_Channel_DPM_Timeout_2						AT%I*  : bool;
	{attribute 'TcLinkTo' := 'TIID^Device 2 (EtherCAT)^Term 1 (EK1200)^Term 4 (EL3446)^I3 Channel^TxPDO Toggle'}
	MDP5001_342_I3_Channel_TxPDO_Toggle_2						AT%I*  : bool;
	{attribute 'TcLinkTo' := 'TIID^Device 2 (EtherCAT)^Term 1 (EK1200)^Term 4 (EL3446)^I3 Channel^Current'}
	MDP5001_342_I3_Channel_Current_2							AT%I*  : REAL;
	{attribute 'TcLinkTo' := 'TIID^Device 2 (EtherCAT)^Term 1 (EK1200)^Term 4 (EL3446)^I3 Channel^Active Power'}
	MDP5001_342_I3_Channel_Active_Power_2						AT%I*  : REAL;
	{attribute 'TcLinkTo' := 'TIID^Device 2 (EtherCAT)^Term 1 (EK1200)^Term 4 (EL3446)^I3 Channel^Apparent Power'}
	MDP5001_342_I3_Channel_Apparent_Power_2					AT%I*  : REAL;
	{attribute 'TcLinkTo' := 'TIID^Device 2 (EtherCAT)^Term 1 (EK1200)^Term 4 (EL3446)^I3 Channel^Reactive Power Fundamental'}
	MDP5001_342_I3_Channel_Reactive_Power_Fundamental_2		AT%I*  : REAL;
	{attribute 'TcLinkTo' := 'TIID^Device 2 (EtherCAT)^Term 1 (EK1200)^Term 4 (EL3446)^I3 Channel^Active Energy'}
	MDP5001_342_I3_Channel_Active_Energy_2					AT%I*  : DINT;	
	{attribute 'TcLinkTo' := 'TIID^Device 2 (EtherCAT)^Term 1 (EK1200)^Term 4 (EL3446)^I4 Channel^Overcurrent'}
	MDP5001_342_I4_Channel_Overcurrent_2						AT%I*  : BOOL;
	{attribute 'TcLinkTo' := 'TIID^Device 2 (EtherCAT)^Term 1 (EK1200)^Term 4 (EL3446)^I4 Channel^Inaccurate Current'}
	MDP5001_342_I4_Channel_Inaccurate_Current_2				AT%I*  : BOOL;
	{attribute 'TcLinkTo' := 'TIID^Device 2 (EtherCAT)^Term 1 (EK1200)^Term 4 (EL3446)^I4 Channel^Current Guard Warning'}
	MDP5001_342_I4_Channel_Current_Guard_Warning_2			AT%I*  : bool;
	{attribute 'TcLinkTo' := 'TIID^Device 2 (EtherCAT)^Term 1 (EK1200)^Term 4 (EL3446)^I4 Channel^Current Guard Error'}
	MDP5001_342_I4_Channel_Current_Guard_Error_2				AT%I*  : bool;
	{attribute 'TcLinkTo' := 'TIID^Device 2 (EtherCAT)^Term 1 (EK1200)^Term 4 (EL3446)^I4 Channel^Apparent Power Guard Warning'}
	MDP5001_342_I4_Channel_Apparent_Power_Guard_Warning_2		AT%I*  : bool;
	{attribute 'TcLinkTo' := 'TIID^Device 2 (EtherCAT)^Term 1 (EK1200)^Term 4 (EL3446)^I4 Channel^Apparent Power Guard Error'}
	MDP5001_342_I4_Channel_Apparent_Power_Guard_Error_2		AT%I*  : bool;
	{attribute 'TcLinkTo' := 'TIID^Device 2 (EtherCAT)^Term 1 (EK1200)^Term 4 (EL3446)^I4 Channel^Active Power Guard Warning'}
	MDP5001_342_I4_Channel_Active_Power_Guard_Warning_2		AT%I*  : bool;
	{attribute 'TcLinkTo' := 'TIID^Device 2 (EtherCAT)^Term 1 (EK1200)^Term 4 (EL3446)^I4 Channel^Active Power Guard Error'}
	MDP5001_342_I4_Channel_Active_Power_Guard_Error_2			AT%I*  : bool;
	{attribute 'TcLinkTo' := 'TIID^Device 2 (EtherCAT)^Term 1 (EK1200)^Term 4 (EL3446)^I4 Channel^Reactive Power Guard Warning'}
	MDP5001_342_I4_Channel_Reactive_Power_Guard_Warning_2		AT%I*  : bool;
	{attribute 'TcLinkTo' := 'TIID^Device 2 (EtherCAT)^Term 1 (EK1200)^Term 4 (EL3446)^I4 Channel^Reactive Power Guard Error'}
	MDP5001_342_I4_Channel_Reactive_Power_Guard_Error_2		AT%I*  : bool;
	{attribute 'TcLinkTo' := 'TIID^Device 2 (EtherCAT)^Term 1 (EK1200)^Term 4 (EL3446)^I4 Channel^DPM Inaccurate'}
	MDP5001_342_I4_Channel_DPM_Inaccurate_2					AT%I*  : bool;
	{attribute 'TcLinkTo' := 'TIID^Device 2 (EtherCAT)^Term 1 (EK1200)^Term 4 (EL3446)^I4 Channel^DPM Timeout'}
	MDP5001_342_I4_Channel_DPM_Timeout_2						AT%I*  : bool;
	{attribute 'TcLinkTo' := 'TIID^Device 2 (EtherCAT)^Term 1 (EK1200)^Term 4 (EL3446)^I4 Channel^TxPDO Toggle'}
	MDP5001_342_I4_Channel_TxPDO_Toggle_2						AT%I*  : bool;
	{attribute 'TcLinkTo' := 'TIID^Device 2 (EtherCAT)^Term 1 (EK1200)^Term 4 (EL3446)^I4 Channel^Current'}
	MDP5001_342_I4_Channel_Current_2							AT%I*  : REAL;
	{attribute 'TcLinkTo' := 'TIID^Device 2 (EtherCAT)^Term 1 (EK1200)^Term 4 (EL3446)^I4 Channel^Active Power'}
	MDP5001_342_I4_Channel_Active_Power_2						AT%I*  : REAL;
	{attribute 'TcLinkTo' := 'TIID^Device 2 (EtherCAT)^Term 1 (EK1200)^Term 4 (EL3446)^I4 Channel^Apparent Power'}
	MDP5001_342_I4_Channel_Apparent_Power_2					AT%I*  : REAL;
	{attribute 'TcLinkTo' := 'TIID^Device 2 (EtherCAT)^Term 1 (EK1200)^Term 4 (EL3446)^I4 Channel^Reactive Power Fundamental'}
	MDP5001_342_I4_Channel_Reactive_Power_Fundamental_2		AT%I*  : REAL;
	{attribute 'TcLinkTo' := 'TIID^Device 2 (EtherCAT)^Term 1 (EK1200)^Term 4 (EL3446)^I4 Channel^Active Energy'}
	MDP5001_342_I4_Channel_Active_Energy_2					AT%I*  : DINT;
	{attribute 'TcLinkTo' := 'TIID^Device 2 (EtherCAT)^Term 1 (EK1200)^Term 4 (EL3446)^I5 Channel^Overcurrent'}
	MDP5001_342_I5_Channel_Overcurrent_2						AT%I*  : BOOL;
	{attribute 'TcLinkTo' := 'TIID^Device 2 (EtherCAT)^Term 1 (EK1200)^Term 4 (EL3446)^I5 Channel^Inaccurate Current'}
	MDP5001_342_I5_Channel_Inaccurate_Current_2				AT%I*  : BOOL;
	{attribute 'TcLinkTo' := 'TIID^Device 2 (EtherCAT)^Term 1 (EK1200)^Term 4 (EL3446)^I5 Channel^Current Guard Warning'}
	MDP5001_342_I5_Channel_Current_Guard_Warning_2			AT%I*  : bool;
	{attribute 'TcLinkTo' := 'TIID^Device 2 (EtherCAT)^Term 1 (EK1200)^Term 4 (EL3446)^I5 Channel^Current Guard Error'}
	MDP5001_342_I5_Channel_Current_Guard_Error_2				AT%I*  : bool;
	{attribute 'TcLinkTo' := 'TIID^Device 2 (EtherCAT)^Term 1 (EK1200)^Term 4 (EL3446)^I5 Channel^Apparent Power Guard Warning'}
	MDP5001_342_I5_Channel_Apparent_Power_Guard_Warning_2		AT%I*  : bool;
	{attribute 'TcLinkTo' := 'TIID^Device 2 (EtherCAT)^Term 1 (EK1200)^Term 4 (EL3446)^I5 Channel^Apparent Power Guard Error'}
	MDP5001_342_I5_Channel_Apparent_Power_Guard_Error_2		AT%I*  : bool;
	{attribute 'TcLinkTo' := 'TIID^Device 2 (EtherCAT)^Term 1 (EK1200)^Term 4 (EL3446)^I5 Channel^Active Power Guard Warning'}
	MDP5001_342_I5_Channel_Active_Power_Guard_Warning_2		AT%I*  : bool;
	{attribute 'TcLinkTo' := 'TIID^Device 2 (EtherCAT)^Term 1 (EK1200)^Term 4 (EL3446)^I5 Channel^Active Power Guard Error'}
	MDP5001_342_I5_Channel_Active_Power_Guard_Error_2			AT%I*  : bool;
	{attribute 'TcLinkTo' := 'TIID^Device 2 (EtherCAT)^Term 1 (EK1200)^Term 4 (EL3446)^I5 Channel^Reactive Power Guard Warning'}
	MDP5001_342_I5_Channel_Reactive_Power_Guard_Warning_2		AT%I*  : bool;
	{attribute 'TcLinkTo' := 'TIID^Device 2 (EtherCAT)^Term 1 (EK1200)^Term 4 (EL3446)^I5 Channel^Reactive Power Guard Error'}
	MDP5001_342_I5_Channel_Reactive_Power_Guard_Error_2		AT%I*  : bool;
	{attribute 'TcLinkTo' := 'TIID^Device 2 (EtherCAT)^Term 1 (EK1200)^Term 4 (EL3446)^I5 Channel^DPM Inaccurate'}
	MDP5001_342_I5_Channel_DPM_Inaccurate_2					AT%I*  : bool;
	{attribute 'TcLinkTo' := 'TIID^Device 2 (EtherCAT)^Term 1 (EK1200)^Term 4 (EL3446)^I5 Channel^DPM Timeout'}
	MDP5001_342_I5_Channel_DPM_Timeout_2						AT%I*  : bool;
	{attribute 'TcLinkTo' := 'TIID^Device 2 (EtherCAT)^Term 1 (EK1200)^Term 4 (EL3446)^I5 Channel^TxPDO Toggle'}
	MDP5001_342_I5_Channel_TxPDO_Toggle_2						AT%I*  : bool;
	{attribute 'TcLinkTo' := 'TIID^Device 2 (EtherCAT)^Term 1 (EK1200)^Term 4 (EL3446)^I5 Channel^Current'}
	MDP5001_342_I5_Channel_Current_2							AT%I*  : REAL;
	{attribute 'TcLinkTo' := 'TIID^Device 2 (EtherCAT)^Term 1 (EK1200)^Term 4 (EL3446)^I5 Channel^Active Power'}
	MDP5001_342_I5_Channel_Active_Power_2						AT%I*  : REAL;
	{attribute 'TcLinkTo' := 'TIID^Device 2 (EtherCAT)^Term 1 (EK1200)^Term 4 (EL3446)^I5 Channel^Apparent Power'}
	MDP5001_342_I5_Channel_Apparent_Power_2					AT%I*  : REAL;
	{attribute 'TcLinkTo' := 'TIID^Device 2 (EtherCAT)^Term 1 (EK1200)^Term 4 (EL3446)^I5 Channel^Reactive Power Fundamental'}
	MDP5001_342_I5_Channel_Reactive_Power_Fundamental_2		AT%I*  : REAL;
	{attribute 'TcLinkTo' := 'TIID^Device 2 (EtherCAT)^Term 1 (EK1200)^Term 4 (EL3446)^I5 Channel^Active Energy'}
	MDP5001_342_I5_Channel_Active_Energy_2					AT%I*  : DINT;
	{attribute 'TcLinkTo' := 'TIID^Device 2 (EtherCAT)^Term 1 (EK1200)^Term 4 (EL3446)^I6 Channel^Overcurrent'}
	MDP5001_342_I6_Channel_Overcurrent_2						AT%I*  : BOOL;
	{attribute 'TcLinkTo' := 'TIID^Device 2 (EtherCAT)^Term 1 (EK1200)^Term 4 (EL3446)^I6 Channel^Inaccurate Current'}
	MDP5001_342_I6_Channel_Inaccurate_Current_2				AT%I*  : BOOL;
	{attribute 'TcLinkTo' := 'TIID^Device 2 (EtherCAT)^Term 1 (EK1200)^Term 4 (EL3446)^I6 Channel^Current Guard Warning'}
	MDP5001_342_I6_Channel_Current_Guard_Warning_2			AT%I*  : bool;
	{attribute 'TcLinkTo' := 'TIID^Device 2 (EtherCAT)^Term 1 (EK1200)^Term 4 (EL3446)^I6 Channel^Current Guard Error'}
	MDP5001_342_I6_Channel_Current_Guard_Error_2				AT%I*  : bool;
	{attribute 'TcLinkTo' := 'TIID^Device 2 (EtherCAT)^Term 1 (EK1200)^Term 4 (EL3446)^I6 Channel^Apparent Power Guard Warning'}
	MDP5001_342_I6_Channel_Apparent_Power_Guard_Warning_2		AT%I*  : bool;
	{attribute 'TcLinkTo' := 'TIID^Device 2 (EtherCAT)^Term 1 (EK1200)^Term 4 (EL3446)^I6 Channel^Apparent Power Guard Error'}
	MDP5001_342_I6_Channel_Apparent_Power_Guard_Error_2		AT%I*  : bool;
	{attribute 'TcLinkTo' := 'TIID^Device 2 (EtherCAT)^Term 1 (EK1200)^Term 4 (EL3446)^I6 Channel^Active Power Guard Warning'}
	MDP5001_342_I6_Channel_Active_Power_Guard_Warning_2		AT%I*  : bool;
	{attribute 'TcLinkTo' := 'TIID^Device 2 (EtherCAT)^Term 1 (EK1200)^Term 4 (EL3446)^I6 Channel^Active Power Guard Error'}
	MDP5001_342_I6_Channel_Active_Power_Guard_Error_2			AT%I*  : bool;
	{attribute 'TcLinkTo' := 'TIID^Device 2 (EtherCAT)^Term 1 (EK1200)^Term 4 (EL3446)^I6 Channel^Reactive Power Guard Warning'}
	MDP5001_342_I6_Channel_Reactive_Power_Guard_Warning_2		AT%I*  : bool;
	{attribute 'TcLinkTo' := 'TIID^Device 2 (EtherCAT)^Term 1 (EK1200)^Term 4 (EL3446)^I6 Channel^Reactive Power Guard Error'}
	MDP5001_342_I6_Channel_Reactive_Power_Guard_Error_2		AT%I*  : bool;
	{attribute 'TcLinkTo' := 'TIID^Device 2 (EtherCAT)^Term 1 (EK1200)^Term 4 (EL3446)^I6 Channel^DPM Inaccurate'}
	MDP5001_342_I6_Channel_DPM_Inaccurate_2					AT%I*  : bool;
	{attribute 'TcLinkTo' := 'TIID^Device 2 (EtherCAT)^Term 1 (EK1200)^Term 4 (EL3446)^I6 Channel^DPM Timeout'}
	MDP5001_342_I6_Channel_DPM_Timeout_2						AT%I*  : bool;
	{attribute 'TcLinkTo' := 'TIID^Device 2 (EtherCAT)^Term 1 (EK1200)^Term 4 (EL3446)^I6 Channel^TxPDO Toggle'}
	MDP5001_342_I6_Channel_TxPDO_Toggle_2						AT%I*  : bool;
	{attribute 'TcLinkTo' := 'TIID^Device 2 (EtherCAT)^Term 1 (EK1200)^Term 4 (EL3446)^I6 Channel^Current'}
	MDP5001_342_I6_Channel_Current_2							AT%I*  : REAL;
	{attribute 'TcLinkTo' := 'TIID^Device 2 (EtherCAT)^Term 1 (EK1200)^Term 4 (EL3446)^I6 Channel^Active Power'}
	MDP5001_342_I6_Channel_Active_Power_2						AT%I*  : REAL;
	{attribute 'TcLinkTo' := 'TIID^Device 2 (EtherCAT)^Term 1 (EK1200)^Term 4 (EL3446)^I6 Channel^Apparent Power'}
	MDP5001_342_I6_Channel_Apparent_Power_2					AT%I*  : REAL;
	{attribute 'TcLinkTo' := 'TIID^Device 2 (EtherCAT)^Term 1 (EK1200)^Term 4 (EL3446)^I6 Channel^Reactive Power Fundamental'}
	MDP5001_342_I6_Channel_Reactive_Power_Fundamental_2		AT%I*  : REAL;
	{attribute 'TcLinkTo' := 'TIID^Device 2 (EtherCAT)^Term 1 (EK1200)^Term 4 (EL3446)^I6 Channel^Active Energy'}
	MDP5001_342_I6_Channel_Active_Energy_2					AT%I*  : DINT;	
	
	{attribute 'TcLinkTo' := 'TIID^Device 2 (EtherCAT)^Term 1 (EK1200)^Term 4 (EL3446)^DPM Variant Value In^TxPDO Toggle'}
	MDP5001_342_DPM_Variant_Value_In_TxPDO_Toggle_2			AT%I*  : BOOL;
	{attribute 'TcLinkTo' := 'TIID^Device 2 (EtherCAT)^Term 1 (EK1200)^Term 4 (EL3446)^DPM Variant Value In^Index 1 REAL'}
	MDP5001_342_DPM_Variant_Value_In_Index_1_REAL_2			AT%I*  : UINT;
	{attribute 'TcLinkTo' := 'TIID^Device 2 (EtherCAT)^Term 1 (EK1200)^Term 4 (EL3446)^DPM Variant Value In^Value 1 REAL'}
	MDP5001_342_DPM_Variant_Value_In_Value_1_REAL_2			AT%I*  : REAL;
	{attribute 'TcLinkTo' := 'TIID^Device 2 (EtherCAT)^Term 1 (EK1200)^Term 4 (EL3446)^DPM Variant Value In^Index 2 REAL'}
	MDP5001_342_DPM_Variant_Value_In_Index_2_REAL_2			AT%I*  : UINT;
	{attribute 'TcLinkTo' := 'TIID^Device 2 (EtherCAT)^Term 1 (EK1200)^Term 4 (EL3446)^DPM Variant Value In^Value 2 REAL'}
	MDP5001_342_DPM_Variant_Value_In_Value_2_REAL_2			AT%I*  : REAL;
	{attribute 'TcLinkTo' := 'TIID^Device 2 (EtherCAT)^Term 1 (EK1200)^Term 4 (EL3446)^DPM Variant Value In^Index 3 REAL'}
	MDP5001_342_DPM_Variant_Value_In_Index_3_REAL_2			AT%I*  : UINT;
	{attribute 'TcLinkTo' := 'TIID^Device 2 (EtherCAT)^Term 1 (EK1200)^Term 4 (EL3446)^DPM Variant Value In^Value 3 REAL'}
	MDP5001_342_DPM_Variant_Value_In_Value_3_REAL_2			AT%I*  : REAL;
	{attribute 'TcLinkTo' := 'TIID^Device 2 (EtherCAT)^Term 1 (EK1200)^Term 4 (EL3446)^DPM Variant Value In^Index 4 ULINT'}
	MDP5001_342_DPM_Variant_Value_In_Index_4_ULINT_2			AT%I*  : UINT;
	{attribute 'TcLinkTo' := 'TIID^Device 2 (EtherCAT)^Term 1 (EK1200)^Term 4 (EL3446)^DPM Variant Value In^Value 4 ULINT'}
	MDP5001_342_DPM_Variant_Value_In_Value_4_ULINT_2			AT%I*  : ULINT;

	{attribute 'TcLinkTo' := 'TIID^Device 2 (EtherCAT)^Term 1 (EK1200)^Term 4 (EL3446)^DPM Variant Value Out^Index 1 REAL'}
	MDP5001_342_DPM_Variant_Value_Out_Index_1_REAL_2	AT%Q* : UINT;
	{attribute 'TcLinkTo' := 'TIID^Device 2 (EtherCAT)^Term 1 (EK1200)^Term 4 (EL3446)^DPM Variant Value Out^Index 2 REAL'}
	MDP5001_342_DPM_Variant_Value_Out_Index_2_REAL_2	AT%Q* : UINT;
	{attribute 'TcLinkTo' := 'TIID^Device 2 (EtherCAT)^Term 1 (EK1200)^Term 4 (EL3446)^DPM Variant Value Out^Index 3 REAL'}
	MDP5001_342_DPM_Variant_Value_Out_Index_3_REAL_2	AT%Q* : UINT;
	{attribute 'TcLinkTo' := 'TIID^Device 2 (EtherCAT)^Term 1 (EK1200)^Term 4 (EL3446)^DPM Variant Value Out^Index 4 ULINT'}
	MDP5001_342_DPM_Variant_Value_Out_Index_4_ULINT_2	AT%Q* : UINT;
	{attribute 'TcLinkTo' := 'TIID^Device 2 (EtherCAT)^Term 1 (EK1200)^Term 4 (EL3446)^DPM Data^Data 1'}
	MDP5001_342_DPM_Data_Data_1_2						AT%Q* : UDINT;
	{attribute 'TcLinkTo' := 'TIID^Device 2 (EtherCAT)^Term 1 (EK1200)^Term 4 (EL3446)^DPM Data^Data 2'}
	MDP5001_342_DPM_Data_Data_2_2						AT%Q* : UDINT;
	{attribute 'TcLinkTo' := 'TIID^Device 2 (EtherCAT)^Term 1 (EK1200)^Term 4 (EL3446)^DPM Data^Data 3'}
	MDP5001_342_DPM_Data_Data_3_2						AT%Q* : UDINT;
	{attribute 'TcLinkTo' := 'TIID^Device 2 (EtherCAT)^Term 1 (EK1200)^Term 4 (EL3446)^DPM Data^Data 4'}
	MDP5001_342_DPM_Data_Data_4_2						AT%Q* : UDINT;
	{attribute 'TcLinkTo' := 'TIID^Device 2 (EtherCAT)^Term 1 (EK1200)^Term 4 (EL3446)^DPM Data^Data 5'}
	MDP5001_342_DPM_Data_Data_5_2						AT%Q* : UDINT;
	{attribute 'TcLinkTo' := 'TIID^Device 2 (EtherCAT)^Term 1 (EK1200)^Term 4 (EL3446)^DPM Data^Data 6'}
	MDP5001_342_DPM_Data_Data_6_2						AT%Q* : UDINT;
	{attribute 'TcLinkTo' := 'TIID^Device 2 (EtherCAT)^Term 1 (EK1200)^Term 4 (EL3446)^DPM Data^Data 7'}
	MDP5001_342_DPM_Data_Data_7_2						AT%Q* : UDINT;
	{attribute 'TcLinkTo' := 'TIID^Device 2 (EtherCAT)^Term 1 (EK1200)^Term 4 (EL3446)^DPM Data^Data 8'}
	MDP5001_342_DPM_Data_Data_8_2						AT%Q* : UDINT;
	{attribute 'TcLinkTo' := 'TIID^Device 2 (EtherCAT)^Term 1 (EK1200)^Term 4 (EL3446)^DPM Data^Data 9'}
	MDP5001_342_DPM_Data_Data_9_2						AT%Q* : UDINT;
	{attribute 'TcLinkTo' := 'TIID^Device 2 (EtherCAT)^Term 1 (EK1200)^Term 4 (EL3446)^DPM Data^Data 10'}
	MDP5001_342_DPM_Data_Data_10_2					AT%Q* : UDINT;
	{attribute 'TcLinkTo' := 'TIID^Device 2 (EtherCAT)^Term 1 (EK1200)^Term 4 (EL3446)^DPM Data^Data 11'}
	MDP5001_342_DPM_Data_Data_11_2					AT%Q* : UDINT;
	{attribute 'TcLinkTo' := 'TIID^Device 2 (EtherCAT)^Term 1 (EK1200)^Term 4 (EL3446)^DPM Data^Data 12'}
	MDP5001_342_DPM_Data_Data_12_2					AT%Q* : UDINT;
	{attribute 'TcLinkTo' := 'TIID^Device 2 (EtherCAT)^Term 1 (EK1200)^Term 4 (EL3446)^DPM Data^Data 13'}
	MDP5001_342_DPM_Data_Data_13_2					AT%Q* : UDINT;
	{attribute 'TcLinkTo' := 'TIID^Device 2 (EtherCAT)^Term 1 (EK1200)^Term 4 (EL3446)^DPM Data^Data 14'}
	MDP5001_342_DPM_Data_Data_14_2					AT%Q* : UDINT;
	{attribute 'TcLinkTo' := 'TIID^Device 2 (EtherCAT)^Term 1 (EK1200)^Term 4 (EL3446)^DPM Data^Data 15'}
	MDP5001_342_DPM_Data_Data_15_2					AT%Q* : UDINT;
	{attribute 'TcLinkTo' := 'TIID^Device 2 (EtherCAT)^Term 1 (EK1200)^Term 4 (EL3446)^DPM Data^Data 16'}
	MDP5001_342_DPM_Data_Data_16_2					AT%Q* : UDINT;
	{attribute 'TcLinkTo' := 'TIID^Device 2 (EtherCAT)^Term 1 (EK1200)^Term 4 (EL3446)^DPM Data^Data 17'}
	MDP5001_342_DPM_Data_Data_17_2					AT%Q* : UDINT;
	{attribute 'TcLinkTo' := 'TIID^Device 2 (EtherCAT)^Term 1 (EK1200)^Term 4 (EL3446)^DPM Data^Data 18'}
	MDP5001_342_DPM_Data_Data_18_2					AT%Q* : UDINT;
	{attribute 'TcLinkTo' := 'TIID^Device 2 (EtherCAT)^Term 1 (EK1200)^Term 4 (EL3446)^DPM Data^Data 19'}
	MDP5001_342_DPM_Data_Data_19_2					AT%Q* : UDINT;
	{attribute 'TcLinkTo' := 'TIID^Device 2 (EtherCAT)^Term 1 (EK1200)^Term 4 (EL3446)^DPM Data^Data 20'}
	MDP5001_342_DPM_Data_Data_20_2					AT%Q* : UDINT;

END_VAR

// copy HW Data to FBs accordingly

//EL3443
prgEM.stEL3443_IO_1.MDP5001_341_Input.MDP5001_341_L1_Status_Voltage_Sign_Bit 		:= MDP5001_341_L1_Status_Voltage_Sign_Bit;
prgEM.stEL3443_IO_1.MDP5001_341_Input.MDP5001_341_L1_Status_Overvoltage			:= MDP5001_341_L1_Status_Overvoltage;
prgEM.stEL3443_IO_1.MDP5001_341_Input.MDP5001_341_L1_Status_Overcurrent			:= MDP5001_341_L1_Status_Overcurrent;
prgEM.stEL3443_IO_1.MDP5001_341_Input.MDP5001_341_L1_Status_Inaccurate_Voltage	:= MDP5001_341_L1_Status_Inaccurate_Voltage;
prgEM.stEL3443_IO_1.MDP5001_341_Input.MDP5001_341_L1_Status_Inaccurate_Current	:= MDP5001_341_L1_Status_Inaccurate_Current;
prgEM.stEL3443_IO_1.MDP5001_341_Input.MDP5001_341_L1_Status_Voltage_Guard_Warning	:= MDP5001_341_L1_Status_Voltage_Guard_Warning;
prgEM.stEL3443_IO_1.MDP5001_341_Input.MDP5001_341_L1_Status_Voltage_Guard_Error	:= MDP5001_341_L1_Status_Voltage_Guard_Error;
prgEM.stEL3443_IO_1.MDP5001_341_Input.MDP5001_341_L1_Status_Current_Guard_Warning	:= MDP5001_341_L1_Status_Current_Guard_Warning;
prgEM.stEL3443_IO_1.MDP5001_341_Input.MDP5001_341_L1_Status_Current_Guard_Error	:= MDP5001_341_L1_Status_Current_Guard_Error;
prgEM.stEL3443_IO_1.MDP5001_341_Input.MDP5001_341_L1_Status_TxPDO_Toggle			:= MDP5001_341_L1_Status_TxPDO_Toggle;
prgEM.stEL3443_IO_1.MDP5001_341_Input.MDP5001_341_L1_Basic_Voltage				:= MDP5001_341_L1_Basic_Voltage;
prgEM.stEL3443_IO_1.MDP5001_341_Input.MDP5001_341_L1_Basic_Current				:= MDP5001_341_L1_Basic_Current;
prgEM.stEL3443_IO_1.MDP5001_341_Input.MDP5001_341_L1_Power_Active_Power			:= MDP5001_341_L1_Power_Active_Power;
prgEM.stEL3443_IO_1.MDP5001_341_Input.MDP5001_341_L1_Power_Apparent_Power			:= MDP5001_341_L1_Power_Apparent_Power;
prgEM.stEL3443_IO_1.MDP5001_341_Input.MDP5001_341_L1_Power_Reactive_Power			:= MDP5001_341_L1_Power_Reactive_Power;
prgEM.stEL3443_IO_1.MDP5001_341_Input.MDP5001_341_L1_Power_Power_Factor			:= MDP5001_341_L1_Power_Power_Factor;
prgEM.stEL3443_IO_1.MDP5001_341_Input.MDP5001_341_L2_Status_Voltage_Sign_Bit 		:= MDP5001_341_L2_Status_Voltage_Sign_Bit;
prgEM.stEL3443_IO_1.MDP5001_341_Input.MDP5001_341_L2_Status_Overvoltage			:= MDP5001_341_L2_Status_Overvoltage;
prgEM.stEL3443_IO_1.MDP5001_341_Input.MDP5001_341_L2_Status_Overcurrent			:= MDP5001_341_L2_Status_Overcurrent;
prgEM.stEL3443_IO_1.MDP5001_341_Input.MDP5001_341_L2_Status_Inaccurate_Voltage	:= MDP5001_341_L2_Status_Inaccurate_Voltage;
prgEM.stEL3443_IO_1.MDP5001_341_Input.MDP5001_341_L2_Status_Inaccurate_Current	:= MDP5001_341_L2_Status_Inaccurate_Current;
prgEM.stEL3443_IO_1.MDP5001_341_Input.MDP5001_341_L2_Status_Voltage_Guard_Warning	:= MDP5001_341_L2_Status_Voltage_Guard_Warning;
prgEM.stEL3443_IO_1.MDP5001_341_Input.MDP5001_341_L2_Status_Voltage_Guard_Error	:= MDP5001_341_L2_Status_Voltage_Guard_Error;
prgEM.stEL3443_IO_1.MDP5001_341_Input.MDP5001_341_L2_Status_Current_Guard_Warning	:= MDP5001_341_L2_Status_Current_Guard_Warning;
prgEM.stEL3443_IO_1.MDP5001_341_Input.MDP5001_341_L2_Status_Current_Guard_Error	:= MDP5001_341_L2_Status_Current_Guard_Error;
prgEM.stEL3443_IO_1.MDP5001_341_Input.MDP5001_341_L2_Status_TxPDO_Toggle			:= MDP5001_341_L2_Status_TxPDO_Toggle;
prgEM.stEL3443_IO_1.MDP5001_341_Input.MDP5001_341_L2_Basic_Voltage				:= MDP5001_341_L2_Basic_Voltage;
prgEM.stEL3443_IO_1.MDP5001_341_Input.MDP5001_341_L2_Basic_Current				:= MDP5001_341_L2_Basic_Current;
prgEM.stEL3443_IO_1.MDP5001_341_Input.MDP5001_341_L2_Power_Active_Power			:= MDP5001_341_L2_Power_Active_Power;
prgEM.stEL3443_IO_1.MDP5001_341_Input.MDP5001_341_L2_Power_Apparent_Power			:= MDP5001_341_L2_Power_Apparent_Power;
prgEM.stEL3443_IO_1.MDP5001_341_Input.MDP5001_341_L2_Power_Reactive_Power			:= MDP5001_341_L2_Power_Reactive_Power;
prgEM.stEL3443_IO_1.MDP5001_341_Input.MDP5001_341_L2_Power_Power_Factor			:= MDP5001_341_L2_Power_Power_Factor;
prgEM.stEL3443_IO_1.MDP5001_341_Input.MDP5001_341_L3_Status_Voltage_Sign_Bit 		:= MDP5001_341_L3_Status_Voltage_Sign_Bit;
prgEM.stEL3443_IO_1.MDP5001_341_Input.MDP5001_341_L3_Status_Overvoltage			:= MDP5001_341_L3_Status_Overvoltage;
prgEM.stEL3443_IO_1.MDP5001_341_Input.MDP5001_341_L3_Status_Overcurrent			:= MDP5001_341_L3_Status_Overcurrent;
prgEM.stEL3443_IO_1.MDP5001_341_Input.MDP5001_341_L3_Status_Inaccurate_Voltage	:= MDP5001_341_L3_Status_Inaccurate_Voltage;
prgEM.stEL3443_IO_1.MDP5001_341_Input.MDP5001_341_L3_Status_Inaccurate_Current	:= MDP5001_341_L3_Status_Inaccurate_Current;
prgEM.stEL3443_IO_1.MDP5001_341_Input.MDP5001_341_L3_Status_Voltage_Guard_Warning	:= MDP5001_341_L3_Status_Voltage_Guard_Warning;
prgEM.stEL3443_IO_1.MDP5001_341_Input.MDP5001_341_L3_Status_Voltage_Guard_Error	:= MDP5001_341_L3_Status_Voltage_Guard_Error;
prgEM.stEL3443_IO_1.MDP5001_341_Input.MDP5001_341_L3_Status_Current_Guard_Warning	:= MDP5001_341_L3_Status_Current_Guard_Warning;
prgEM.stEL3443_IO_1.MDP5001_341_Input.MDP5001_341_L3_Status_Current_Guard_Error	:= MDP5001_341_L3_Status_Current_Guard_Error;
prgEM.stEL3443_IO_1.MDP5001_341_Input.MDP5001_341_L3_Status_TxPDO_Toggle			:= MDP5001_341_L3_Status_TxPDO_Toggle;
prgEM.stEL3443_IO_1.MDP5001_341_Input.MDP5001_341_L3_Basic_Voltage				:= MDP5001_341_L3_Basic_Voltage;
prgEM.stEL3443_IO_1.MDP5001_341_Input.MDP5001_341_L3_Basic_Current				:= MDP5001_341_L3_Basic_Current;
prgEM.stEL3443_IO_1.MDP5001_341_Input.MDP5001_341_L3_Power_Active_Power			:= MDP5001_341_L3_Power_Active_Power;
prgEM.stEL3443_IO_1.MDP5001_341_Input.MDP5001_341_L3_Power_Apparent_Power			:= MDP5001_341_L3_Power_Apparent_Power;
prgEM.stEL3443_IO_1.MDP5001_341_Input.MDP5001_341_L3_Power_Reactive_Power			:= MDP5001_341_L3_Power_Reactive_Power;
prgEM.stEL3443_IO_1.MDP5001_341_Input.MDP5001_341_L3_Power_Power_Factor			:= MDP5001_341_L3_Power_Power_Factor;
prgEM.stEL3443_IO_1.MDP5001_341_Input.MDP5001_341_Total_Status_System_State		:= MDP5001_341_Total_Status_System_State  ;	
prgEM.stEL3443_IO_1.MDP5001_341_Input.MDP5001_341_Total_Status_Grid_Direction		:= MDP5001_341_Total_Status_Grid_Direction ;
prgEM.stEL3443_IO_1.MDP5001_341_Input.MDP5001_341_Total_Status_Frequency_Guard_Warning 		:= MDP5001_341_Total_Status_Frequency_Guard_Warning ;
prgEM.stEL3443_IO_1.MDP5001_341_Input.MDP5001_341_Total_Status_Frequency_Guard_Error 			:= MDP5001_341_Total_Status_Frequency_Guard_Error  ;
prgEM.stEL3443_IO_1.MDP5001_341_Input.MDP5001_341_Total_Status_Neutral_Current_Guard_Warning	:= MDP5001_341_Total_Status_Neutral_Current_Guard_Warning ;
prgEM.stEL3443_IO_1.MDP5001_341_Input.MDP5001_341_Total_Status_Neutral_Current_Guard_Error	:= MDP5001_341_Total_Status_Neutral_Current_Guard_Error;
prgEM.stEL3443_IO_1.MDP5001_341_Input.MDP5001_341_Total_Status_Active_Power_Guard_Warning		:= MDP5001_341_Total_Status_Active_Power_Guard_Warning ;
prgEM.stEL3443_IO_1.MDP5001_341_Input.MDP5001_341_Total_Status_Active_Power_Guard_Error		:= MDP5001_341_Total_Status_Active_Power_Guard_Error ;
prgEM.stEL3443_IO_1.MDP5001_341_Input.MDP5001_341_Total_Status_Apparent_Power_Guard_Warning	:= MDP5001_341_Total_Status_Apparent_Power_Guard_Warning ;
prgEM.stEL3443_IO_1.MDP5001_341_Input.MDP5001_341_Total_Status_Apparent_Power_Guard_Error		:= MDP5001_341_Total_Status_Apparent_Power_Guard_Error ;
prgEM.stEL3443_IO_1.MDP5001_341_Input.MDP5001_341_Total_Status_Power_Quality_Guard_Warning	:= MDP5001_341_Total_Status_Power_Quality_Guard_Warning ;
prgEM.stEL3443_IO_1.MDP5001_341_Input.MDP5001_341_Total_Status_Power_Quality_Guard_Error		:= MDP5001_341_Total_Status_Power_Quality_Guard_Error ;
prgEM.stEL3443_IO_1.MDP5001_341_Input.MDP5001_341_Total_Status_TxPDO_State					:= MDP5001_341_Total_Status_TxPDO_State ;
prgEM.stEL3443_IO_1.MDP5001_341_Input.MDP5001_341_Total_Status_TxPDO_Toggle					:= MDP5001_341_Total_Status_TxPDO_Toggle ;
prgEM.stEL3443_IO_1.MDP5001_341_Input.MDP5001_341_Total_Status_Power_Quality_Factor			:= MDP5001_341_Total_Status_Power_Quality_Factor ;
prgEM.stEL3443_IO_1.MDP5001_341_Input.MDP5001_341_Total_Basic_Frequency						:= MDP5001_341_Total_Basic_Frequency;
prgEM.stEL3443_IO_1.MDP5001_341_Input.MDP5001_341_Total_Basic_Power_Factor					:= MDP5001_341_Total_Basic_Power_Factor  ;
prgEM.stEL3443_IO_1.MDP5001_341_Input.MDP5001_341_Total_Basic_Calculated_Neutral_Line_Current	:= MDP5001_341_Total_Basic_Calculated_Neutral_Line_Current ;
prgEM.stEL3443_IO_1.MDP5001_341_Input.MDP5001_341_Total_Variant_Value_In_TxPDO_Toggle			:= MDP5001_341_Total_Variant_Value_In_TxPDO_Toggle ;
prgEM.stEL3443_IO_1.MDP5001_341_Input.MDP5001_341_Total_Variant_Value_In_Index_1_REAL			:= MDP5001_341_Total_Variant_Value_In_Index_1_REAL ;
prgEM.stEL3443_IO_1.MDP5001_341_Input.MDP5001_341_Total_Variant_Value_In_Value_1_REAL			:= MDP5001_341_Total_Variant_Value_In_Value_1_REAL ;
prgEM.stEL3443_IO_1.MDP5001_341_Input.MDP5001_341_Total_Variant_Value_In_Index_2_REAL			:= MDP5001_341_Total_Variant_Value_In_Index_2_REAL ;
prgEM.stEL3443_IO_1.MDP5001_341_Input.MDP5001_341_Total_Variant_Value_In_Value_2_REAL			:= MDP5001_341_Total_Variant_Value_In_Value_2_REAL ;
prgEM.stEL3443_IO_1.MDP5001_341_Input.MDP5001_341_Total_Variant_Value_In_Index_3_REAL			:= MDP5001_341_Total_Variant_Value_In_Index_3_REAL ;
prgEM.stEL3443_IO_1.MDP5001_341_Input.MDP5001_341_Total_Variant_Value_In_Value_3_REAL			:= MDP5001_341_Total_Variant_Value_In_Value_3_REAL ;
prgEM.stEL3443_IO_1.MDP5001_341_Input.MDP5001_341_Total_Variant_Value_In_Index_4_ULINT		:= MDP5001_341_Total_Variant_Value_In_Index_4_ULINT ;
prgEM.stEL3443_IO_1.MDP5001_341_Input.MDP5001_341_Total_Variant_Value_In_Value_4_ULINT		:= MDP5001_341_Total_Variant_Value_In_Value_4_ULINT ;
prgEM.stEL3443_IO_1.MDP5001_341_Input.MDP5001_341_DPM_Data_Data_1			:= MDP5001_341_DPM_Data_Data_1;
prgEM.stEL3443_IO_1.MDP5001_341_Input.MDP5001_341_DPM_Data_Data_2			:= MDP5001_341_DPM_Data_Data_2;
prgEM.stEL3443_IO_1.MDP5001_341_Input.MDP5001_341_DPM_Data_Data_3			:= MDP5001_341_DPM_Data_Data_3;
prgEM.stEL3443_IO_1.MDP5001_341_Input.MDP5001_341_DPM_Data_Data_4			:= MDP5001_341_DPM_Data_Data_4;
prgEM.stEL3443_IO_1.MDP5001_341_Input.MDP5001_341_DPM_Data_Data_5			:= MDP5001_341_DPM_Data_Data_5;
prgEM.stEL3443_IO_1.MDP5001_341_Input.MDP5001_341_DPM_Data_Data_6			:= MDP5001_341_DPM_Data_Data_6;
prgEM.stEL3443_IO_1.MDP5001_341_Input.MDP5001_341_DPM_Data_Data_7			:= MDP5001_341_DPM_Data_Data_7;
prgEM.stEL3443_IO_1.MDP5001_341_Input.MDP5001_341_DPM_Data_Data_8			:= MDP5001_341_DPM_Data_Data_8;
prgEM.stEL3443_IO_1.MDP5001_341_Input.MDP5001_341_DPM_Data_Data_9			:= MDP5001_341_DPM_Data_Data_9;
prgEM.stEL3443_IO_1.MDP5001_341_Input.MDP5001_341_DPM_Data_Data_10		:= MDP5001_341_DPM_Data_Data_10;
prgEM.stEL3443_IO_1.MDP5001_341_Input.MDP5001_341_DPM_Data_Data_11		:= MDP5001_341_DPM_Data_Data_11;
prgEM.stEL3443_IO_1.MDP5001_341_Input.MDP5001_341_DPM_Data_Data_12		:= MDP5001_341_DPM_Data_Data_12;
prgEM.stEL3443_IO_1.MDP5001_341_Input.MDP5001_341_DPM_Data_Data_13		:= MDP5001_341_DPM_Data_Data_13;
prgEM.stEL3443_IO_1.MDP5001_341_Input.MDP5001_341_DPM_Data_Data_14		:= MDP5001_341_DPM_Data_Data_14;
prgEM.stEL3443_IO_1.MDP5001_341_Input.MDP5001_341_DPM_Data_Data_15		:= MDP5001_341_DPM_Data_Data_15;
prgEM.stEL3443_IO_1.MDP5001_341_Input.MDP5001_341_DPM_Data_Data_16		:= MDP5001_341_DPM_Data_Data_16;
prgEM.stEL3443_IO_1.MDP5001_341_Input.MDP5001_341_DPM_Data_Data_17		:= MDP5001_341_DPM_Data_Data_17;
prgEM.stEL3443_IO_1.MDP5001_341_Input.MDP5001_341_DPM_Data_Data_18		:= MDP5001_341_DPM_Data_Data_18;
prgEM.stEL3443_IO_1.MDP5001_341_Input.MDP5001_341_DPM_Data_Data_19		:= MDP5001_341_DPM_Data_Data_19;
prgEM.stEL3443_IO_1.MDP5001_341_Input.MDP5001_341_DPM_Data_Data_20		:= MDP5001_341_DPM_Data_Data_20;
MDP5001_341_Total_Variant_Value_Out_Index_1_REAL	:= prgEM.stEL3443_IO_1.MDP5001_341_Output.MDP5001_341_Total_Variant_Value_Out_Index_1_REAL;
MDP5001_341_Total_Variant_Value_Out_Index_2_REAL	:= prgEM.stEL3443_IO_1.MDP5001_341_Output.MDP5001_341_Total_Variant_Value_Out_Index_2_REAL;
MDP5001_341_Total_Variant_Value_Out_Index_3_REAL	:= prgEM.stEL3443_IO_1.MDP5001_341_Output.MDP5001_341_Total_Variant_Value_Out_Index_3_REAL;
MDP5001_341_Total_Variant_Value_Out_Index_4_ULINT	:= prgEM.stEL3443_IO_1.MDP5001_341_Output.MDP5001_341_Total_Variant_Value_Out_Index_4_ULINT;
MDP5001_341_Total_Interval_Reset_Interval			:= prgEM.stEL3443_IO_1.MDP5001_341_Output.MDP5001_341_Total_Interval_Reset_Interval;


//EL3443

prgEM.stEL3443_IO_2.MDP5001_341_Input.MDP5001_341_L1_Status_Voltage_Sign_Bit 		:= MDP5001_342_L1_Status_Voltage_Sign_Bit;
prgEM.stEL3443_IO_2.MDP5001_341_Input.MDP5001_341_L1_Status_Overvoltage				:= MDP5001_342_L1_Status_Overvoltage;
prgEM.stEL3443_IO_2.MDP5001_341_Input.MDP5001_341_L1_Status_Overcurrent				:= MDP5001_342_L1_Status_Overcurrent;
prgEM.stEL3443_IO_2.MDP5001_341_Input.MDP5001_341_L1_Status_Inaccurate_Voltage		:= MDP5001_342_L1_Status_Inaccurate_Voltage;
prgEM.stEL3443_IO_2.MDP5001_341_Input.MDP5001_341_L1_Status_Inaccurate_Current		:= MDP5001_342_L1_Status_Inaccurate_Current;
prgEM.stEL3443_IO_2.MDP5001_341_Input.MDP5001_341_L1_Status_Voltage_Guard_Warning	:= MDP5001_342_L1_Status_Voltage_Guard_Warning;
prgEM.stEL3443_IO_2.MDP5001_341_Input.MDP5001_341_L1_Status_Voltage_Guard_Error		:= MDP5001_342_L1_Status_Voltage_Guard_Error;
prgEM.stEL3443_IO_2.MDP5001_341_Input.MDP5001_341_L1_Status_Current_Guard_Warning	:= MDP5001_342_L1_Status_Current_Guard_Warning;
prgEM.stEL3443_IO_2.MDP5001_341_Input.MDP5001_341_L1_Status_Current_Guard_Error		:= MDP5001_342_L1_Status_Current_Guard_Error;
prgEM.stEL3443_IO_2.MDP5001_341_Input.MDP5001_341_L1_Status_TxPDO_Toggle			:= MDP5001_342_L1_Status_TxPDO_Toggle;
prgEM.stEL3443_IO_2.MDP5001_341_Input.MDP5001_341_L1_Basic_Voltage					:= MDP5001_342_L1_Basic_Voltage;
prgEM.stEL3443_IO_2.MDP5001_341_Input.MDP5001_341_L1_Basic_Current					:= MDP5001_342_L1_Basic_Current;
prgEM.stEL3443_IO_2.MDP5001_341_Input.MDP5001_341_L1_Power_Active_Power				:= MDP5001_342_L1_Power_Active_Power;
prgEM.stEL3443_IO_2.MDP5001_341_Input.MDP5001_341_L1_Power_Apparent_Power			:= MDP5001_342_L1_Power_Apparent_Power;
prgEM.stEL3443_IO_2.MDP5001_341_Input.MDP5001_341_L1_Power_Reactive_Power			:= MDP5001_342_L1_Power_Reactive_Power;
prgEM.stEL3443_IO_2.MDP5001_341_Input.MDP5001_341_L1_Power_Power_Factor				:= MDP5001_342_L1_Power_Power_Factor;
prgEM.stEL3443_IO_2.MDP5001_341_Input.MDP5001_341_L2_Status_Voltage_Sign_Bit 		:= MDP5001_342_L2_Status_Voltage_Sign_Bit;
prgEM.stEL3443_IO_2.MDP5001_341_Input.MDP5001_341_L2_Status_Overvoltage				:= MDP5001_342_L2_Status_Overvoltage;
prgEM.stEL3443_IO_2.MDP5001_341_Input.MDP5001_341_L2_Status_Overcurrent				:= MDP5001_342_L2_Status_Overcurrent;
prgEM.stEL3443_IO_2.MDP5001_341_Input.MDP5001_341_L2_Status_Inaccurate_Voltage		:= MDP5001_342_L2_Status_Inaccurate_Voltage;
prgEM.stEL3443_IO_2.MDP5001_341_Input.MDP5001_341_L2_Status_Inaccurate_Current		:= MDP5001_342_L2_Status_Inaccurate_Current;
prgEM.stEL3443_IO_2.MDP5001_341_Input.MDP5001_341_L2_Status_Voltage_Guard_Warning	:= MDP5001_342_L2_Status_Voltage_Guard_Warning;
prgEM.stEL3443_IO_2.MDP5001_341_Input.MDP5001_341_L2_Status_Voltage_Guard_Error		:= MDP5001_342_L2_Status_Voltage_Guard_Error;
prgEM.stEL3443_IO_2.MDP5001_341_Input.MDP5001_341_L2_Status_Current_Guard_Warning	:= MDP5001_342_L2_Status_Current_Guard_Warning;
prgEM.stEL3443_IO_2.MDP5001_341_Input.MDP5001_341_L2_Status_Current_Guard_Error		:= MDP5001_342_L2_Status_Current_Guard_Error;
prgEM.stEL3443_IO_2.MDP5001_341_Input.MDP5001_341_L2_Status_TxPDO_Toggle			:= MDP5001_342_L2_Status_TxPDO_Toggle;
prgEM.stEL3443_IO_2.MDP5001_341_Input.MDP5001_341_L2_Basic_Voltage					:= MDP5001_342_L2_Basic_Voltage;
prgEM.stEL3443_IO_2.MDP5001_341_Input.MDP5001_341_L2_Basic_Current					:= MDP5001_342_L2_Basic_Current;
prgEM.stEL3443_IO_2.MDP5001_341_Input.MDP5001_341_L2_Power_Active_Power				:= MDP5001_342_L2_Power_Active_Power;
prgEM.stEL3443_IO_2.MDP5001_341_Input.MDP5001_341_L2_Power_Apparent_Power			:= MDP5001_342_L2_Power_Apparent_Power;
prgEM.stEL3443_IO_2.MDP5001_341_Input.MDP5001_341_L2_Power_Reactive_Power			:= MDP5001_342_L2_Power_Reactive_Power;
prgEM.stEL3443_IO_2.MDP5001_341_Input.MDP5001_341_L2_Power_Power_Factor				:= MDP5001_342_L2_Power_Power_Factor;
prgEM.stEL3443_IO_2.MDP5001_341_Input.MDP5001_341_L3_Status_Voltage_Sign_Bit 		:= MDP5001_342_L3_Status_Voltage_Sign_Bit;
prgEM.stEL3443_IO_2.MDP5001_341_Input.MDP5001_341_L3_Status_Overvoltage				:= MDP5001_342_L3_Status_Overvoltage;
prgEM.stEL3443_IO_2.MDP5001_341_Input.MDP5001_341_L3_Status_Overcurrent				:= MDP5001_342_L3_Status_Overcurrent;
prgEM.stEL3443_IO_2.MDP5001_341_Input.MDP5001_341_L3_Status_Inaccurate_Voltage		:= MDP5001_342_L3_Status_Inaccurate_Voltage;
prgEM.stEL3443_IO_2.MDP5001_341_Input.MDP5001_341_L3_Status_Inaccurate_Current		:= MDP5001_342_L3_Status_Inaccurate_Current;
prgEM.stEL3443_IO_2.MDP5001_341_Input.MDP5001_341_L3_Status_Voltage_Guard_Warning	:= MDP5001_342_L3_Status_Voltage_Guard_Warning;
prgEM.stEL3443_IO_2.MDP5001_341_Input.MDP5001_341_L3_Status_Voltage_Guard_Error		:= MDP5001_342_L3_Status_Voltage_Guard_Error;
prgEM.stEL3443_IO_2.MDP5001_341_Input.MDP5001_341_L3_Status_Current_Guard_Warning	:= MDP5001_342_L3_Status_Current_Guard_Warning;
prgEM.stEL3443_IO_2.MDP5001_341_Input.MDP5001_341_L3_Status_Current_Guard_Error		:= MDP5001_342_L3_Status_Current_Guard_Error;
prgEM.stEL3443_IO_2.MDP5001_341_Input.MDP5001_341_L3_Status_TxPDO_Toggle			:= MDP5001_342_L3_Status_TxPDO_Toggle;
prgEM.stEL3443_IO_2.MDP5001_341_Input.MDP5001_341_L3_Basic_Voltage					:= MDP5001_342_L3_Basic_Voltage;
prgEM.stEL3443_IO_2.MDP5001_341_Input.MDP5001_341_L3_Basic_Current					:= MDP5001_342_L3_Basic_Current;
prgEM.stEL3443_IO_2.MDP5001_341_Input.MDP5001_341_L3_Power_Active_Power				:= MDP5001_342_L3_Power_Active_Power;
prgEM.stEL3443_IO_2.MDP5001_341_Input.MDP5001_341_L3_Power_Apparent_Power			:= MDP5001_342_L3_Power_Apparent_Power;
prgEM.stEL3443_IO_2.MDP5001_341_Input.MDP5001_341_L3_Power_Reactive_Power			:= MDP5001_342_L3_Power_Reactive_Power;
prgEM.stEL3443_IO_2.MDP5001_341_Input.MDP5001_341_L3_Power_Power_Factor				:= MDP5001_342_L3_Power_Power_Factor;
prgEM.stEL3443_IO_2.MDP5001_341_Input.MDP5001_341_Total_Status_System_State			:= MDP5001_342_Total_Status_System_State  ;	
prgEM.stEL3443_IO_2.MDP5001_341_Input.MDP5001_341_Total_Status_Grid_Direction		:= MDP5001_342_Total_Status_Grid_Direction ;
prgEM.stEL3443_IO_2.MDP5001_341_Input.MDP5001_341_Total_Status_Frequency_Guard_Warning 			:= MDP5001_342_Total_Status_Frequency_Guard_Warning ;
prgEM.stEL3443_IO_2.MDP5001_341_Input.MDP5001_341_Total_Status_Frequency_Guard_Error 			:= MDP5001_342_Total_Status_Frequency_Guard_Error  ;
prgEM.stEL3443_IO_2.MDP5001_341_Input.MDP5001_341_Total_Status_Neutral_Current_Guard_Warning	:= MDP5001_342_Total_Status_Neutral_Current_Guard_Warning ;
prgEM.stEL3443_IO_2.MDP5001_341_Input.MDP5001_341_Total_Status_Neutral_Current_Guard_Error		:= MDP5001_342_Total_Status_Neutral_Current_Guard_Error;
prgEM.stEL3443_IO_2.MDP5001_341_Input.MDP5001_341_Total_Status_Active_Power_Guard_Warning		:= MDP5001_342_Total_Status_Active_Power_Guard_Warning ;
prgEM.stEL3443_IO_2.MDP5001_341_Input.MDP5001_341_Total_Status_Active_Power_Guard_Error			:= MDP5001_342_Total_Status_Active_Power_Guard_Error ;
prgEM.stEL3443_IO_2.MDP5001_341_Input.MDP5001_341_Total_Status_Apparent_Power_Guard_Warning		:= MDP5001_342_Total_Status_Apparent_Power_Guard_Warning ;
prgEM.stEL3443_IO_2.MDP5001_341_Input.MDP5001_341_Total_Status_Apparent_Power_Guard_Error		:= MDP5001_342_Total_Status_Apparent_Power_Guard_Error ;
prgEM.stEL3443_IO_2.MDP5001_341_Input.MDP5001_341_Total_Status_Power_Quality_Guard_Warning		:= MDP5001_342_Total_Status_Power_Quality_Guard_Warning ;
prgEM.stEL3443_IO_2.MDP5001_341_Input.MDP5001_341_Total_Status_Power_Quality_Guard_Error		:= MDP5001_342_Total_Status_Power_Quality_Guard_Error ;
prgEM.stEL3443_IO_2.MDP5001_341_Input.MDP5001_341_Total_Status_TxPDO_State						:= MDP5001_342_Total_Status_TxPDO_State ;
prgEM.stEL3443_IO_2.MDP5001_341_Input.MDP5001_341_Total_Status_TxPDO_Toggle						:= MDP5001_342_Total_Status_TxPDO_Toggle ;
prgEM.stEL3443_IO_2.MDP5001_341_Input.MDP5001_341_Total_Status_Power_Quality_Factor				:= MDP5001_342_Total_Status_Power_Quality_Factor ;
prgEM.stEL3443_IO_2.MDP5001_341_Input.MDP5001_341_Total_Basic_Frequency							:= MDP5001_342_Total_Basic_Frequency;
prgEM.stEL3443_IO_2.MDP5001_341_Input.MDP5001_341_Total_Basic_Power_Factor						:= MDP5001_342_Total_Basic_Power_Factor  ;
prgEM.stEL3443_IO_2.MDP5001_341_Input.MDP5001_341_Total_Basic_Calculated_Neutral_Line_Current	:= MDP5001_342_Total_Basic_Calculated_Neutral_Line_Current ;
prgEM.stEL3443_IO_2.MDP5001_341_Input.MDP5001_341_Total_Variant_Value_In_TxPDO_Toggle			:= MDP5001_342_Total_Variant_Value_In_TxPDO_Toggle ;
prgEM.stEL3443_IO_2.MDP5001_341_Input.MDP5001_341_Total_Variant_Value_In_Index_1_REAL			:= MDP5001_342_Total_Variant_Value_In_Index_1_REAL ;
prgEM.stEL3443_IO_2.MDP5001_341_Input.MDP5001_341_Total_Variant_Value_In_Value_1_REAL			:= MDP5001_342_Total_Variant_Value_In_Value_1_REAL ;
prgEM.stEL3443_IO_2.MDP5001_341_Input.MDP5001_341_Total_Variant_Value_In_Index_2_REAL			:= MDP5001_342_Total_Variant_Value_In_Index_2_REAL ;
prgEM.stEL3443_IO_2.MDP5001_341_Input.MDP5001_341_Total_Variant_Value_In_Value_2_REAL			:= MDP5001_342_Total_Variant_Value_In_Value_2_REAL ;
prgEM.stEL3443_IO_2.MDP5001_341_Input.MDP5001_341_Total_Variant_Value_In_Index_3_REAL			:= MDP5001_342_Total_Variant_Value_In_Index_3_REAL ;
prgEM.stEL3443_IO_2.MDP5001_341_Input.MDP5001_341_Total_Variant_Value_In_Value_3_REAL			:= MDP5001_342_Total_Variant_Value_In_Value_3_REAL ;
prgEM.stEL3443_IO_2.MDP5001_341_Input.MDP5001_341_Total_Variant_Value_In_Index_4_ULINT			:= MDP5001_342_Total_Variant_Value_In_Index_4_ULINT ;
prgEM.stEL3443_IO_2.MDP5001_341_Input.MDP5001_341_Total_Variant_Value_In_Value_4_ULINT			:= MDP5001_342_Total_Variant_Value_In_Value_4_ULINT ;
prgEM.stEL3443_IO_2.MDP5001_341_Input.MDP5001_341_DPM_Data_Data_1			:= MDP5001_342_DPM_Data_Data_1;
prgEM.stEL3443_IO_2.MDP5001_341_Input.MDP5001_341_DPM_Data_Data_2			:= MDP5001_342_DPM_Data_Data_2;
prgEM.stEL3443_IO_2.MDP5001_341_Input.MDP5001_341_DPM_Data_Data_3			:= MDP5001_342_DPM_Data_Data_3;
prgEM.stEL3443_IO_2.MDP5001_341_Input.MDP5001_341_DPM_Data_Data_4			:= MDP5001_342_DPM_Data_Data_4;
prgEM.stEL3443_IO_2.MDP5001_341_Input.MDP5001_341_DPM_Data_Data_5			:= MDP5001_342_DPM_Data_Data_5;
prgEM.stEL3443_IO_2.MDP5001_341_Input.MDP5001_341_DPM_Data_Data_6			:= MDP5001_342_DPM_Data_Data_6;
prgEM.stEL3443_IO_2.MDP5001_341_Input.MDP5001_341_DPM_Data_Data_7			:= MDP5001_342_DPM_Data_Data_7;
prgEM.stEL3443_IO_2.MDP5001_341_Input.MDP5001_341_DPM_Data_Data_8			:= MDP5001_342_DPM_Data_Data_8;
prgEM.stEL3443_IO_2.MDP5001_341_Input.MDP5001_341_DPM_Data_Data_9			:= MDP5001_342_DPM_Data_Data_9;
prgEM.stEL3443_IO_2.MDP5001_341_Input.MDP5001_341_DPM_Data_Data_10			:= MDP5001_342_DPM_Data_Data_10;
prgEM.stEL3443_IO_2.MDP5001_341_Input.MDP5001_341_DPM_Data_Data_11			:= MDP5001_342_DPM_Data_Data_11;
prgEM.stEL3443_IO_2.MDP5001_341_Input.MDP5001_341_DPM_Data_Data_12			:= MDP5001_342_DPM_Data_Data_12;
prgEM.stEL3443_IO_2.MDP5001_341_Input.MDP5001_341_DPM_Data_Data_13			:= MDP5001_342_DPM_Data_Data_13;
prgEM.stEL3443_IO_2.MDP5001_341_Input.MDP5001_341_DPM_Data_Data_14			:= MDP5001_342_DPM_Data_Data_14;
prgEM.stEL3443_IO_2.MDP5001_341_Input.MDP5001_341_DPM_Data_Data_15			:= MDP5001_342_DPM_Data_Data_15;
prgEM.stEL3443_IO_2.MDP5001_341_Input.MDP5001_341_DPM_Data_Data_16			:= MDP5001_342_DPM_Data_Data_16;
prgEM.stEL3443_IO_2.MDP5001_341_Input.MDP5001_341_DPM_Data_Data_17			:= MDP5001_342_DPM_Data_Data_17;
prgEM.stEL3443_IO_2.MDP5001_341_Input.MDP5001_341_DPM_Data_Data_18			:= MDP5001_342_DPM_Data_Data_18;
prgEM.stEL3443_IO_2.MDP5001_341_Input.MDP5001_341_DPM_Data_Data_19			:= MDP5001_342_DPM_Data_Data_19;
prgEM.stEL3443_IO_2.MDP5001_341_Input.MDP5001_341_DPM_Data_Data_20			:= MDP5001_342_DPM_Data_Data_20;
MDP5001_342_Total_Variant_Value_Out_Index_1_REAL	:= prgEM.stEL3443_IO_2.MDP5001_341_Output.MDP5001_341_Total_Variant_Value_Out_Index_1_REAL;
MDP5001_342_Total_Variant_Value_Out_Index_2_REAL	:= prgEM.stEL3443_IO_2.MDP5001_341_Output.MDP5001_341_Total_Variant_Value_Out_Index_2_REAL;
MDP5001_342_Total_Variant_Value_Out_Index_3_REAL	:= prgEM.stEL3443_IO_2.MDP5001_341_Output.MDP5001_341_Total_Variant_Value_Out_Index_3_REAL;
MDP5001_342_Total_Variant_Value_Out_Index_4_ULINT	:= prgEM.stEL3443_IO_2.MDP5001_341_Output.MDP5001_341_Total_Variant_Value_Out_Index_4_ULINT;
MDP5001_342_Total_Interval_Reset_Interval			:= prgEM.stEL3443_IO_2.MDP5001_341_Output.MDP5001_341_Total_Interval_Reset_Interval;



// EL3446

prgEM.stEL3446_IO_1.MDP5001_342_Input.MDP5001_342_I1_Channel_Overcurrent					:=	MDP5001_342_I1_Channel_Overcurrent_1;
prgEM.stEL3446_IO_1.MDP5001_342_Input.MDP5001_342_I1_Channel_Inaccurate_Current			:=	MDP5001_342_I1_Channel_Inaccurate_Current_1;
prgEM.stEL3446_IO_1.MDP5001_342_Input.MDP5001_342_I1_Channel_Current_Guard_Warning		:=	MDP5001_342_I1_Channel_Current_Guard_Warning_1;
prgEM.stEL3446_IO_1.MDP5001_342_Input.MDP5001_342_I1_Channel_Current_Guard_Error			:=	MDP5001_342_I1_Channel_Current_Guard_Error_1;
prgEM.stEL3446_IO_1.MDP5001_342_Input.MDP5001_342_I1_Channel_Apparent_Power_Guard_Warning	:=	MDP5001_342_I1_Channel_Apparent_Power_Guard_Warning_1;
prgEM.stEL3446_IO_1.MDP5001_342_Input.MDP5001_342_I1_Channel_Apparent_Power_Guard_Error	:=	MDP5001_342_I1_Channel_Apparent_Power_Guard_Error_1;
prgEM.stEL3446_IO_1.MDP5001_342_Input.MDP5001_342_I1_Channel_Active_Power_Guard_Warning	:=	MDP5001_342_I1_Channel_Active_Power_Guard_Warning_1;
prgEM.stEL3446_IO_1.MDP5001_342_Input.MDP5001_342_I1_Channel_Active_Power_Guard_Error		:=	MDP5001_342_I1_Channel_Active_Power_Guard_Error_1;
prgEM.stEL3446_IO_1.MDP5001_342_Input.MDP5001_342_I1_Channel_Reactive_Power_Guard_Warning	:=	MDP5001_342_I1_Channel_Reactive_Power_Guard_Warning_1;
prgEM.stEL3446_IO_1.MDP5001_342_Input.MDP5001_342_I1_Channel_Reactive_Power_Guard_Error	:=	MDP5001_342_I1_Channel_Reactive_Power_Guard_Error_1;
prgEM.stEL3446_IO_1.MDP5001_342_Input.MDP5001_342_I1_Channel_DPM_Inaccurate				:=	MDP5001_342_I1_Channel_DPM_Inaccurate_1;
prgEM.stEL3446_IO_1.MDP5001_342_Input.MDP5001_342_I1_Channel_DPM_Timeout					:=	MDP5001_342_I1_Channel_DPM_Timeout_1;
prgEM.stEL3446_IO_1.MDP5001_342_Input.MDP5001_342_I1_Channel_TxPDO_Toggle					:=	MDP5001_342_I1_Channel_TxPDO_Toggle_1;
prgEM.stEL3446_IO_1.MDP5001_342_Input.MDP5001_342_I1_Channel_Current						:=	MDP5001_342_I1_Channel_Current_1;
prgEM.stEL3446_IO_1.MDP5001_342_Input.MDP5001_342_I1_Channel_Active_Power					:=	MDP5001_342_I1_Channel_Active_Power_1;
prgEM.stEL3446_IO_1.MDP5001_342_Input.MDP5001_342_I1_Channel_Apparent_Power				:=	MDP5001_342_I1_Channel_Apparent_Power_1;
prgEM.stEL3446_IO_1.MDP5001_342_Input.MDP5001_342_I1_Channel_Reactive_Power_Fundamental	:=	MDP5001_342_I1_Channel_Reactive_Power_Fundamental_1;
prgEM.stEL3446_IO_1.MDP5001_342_Input.MDP5001_342_I1_Channel_Active_Energy				:=	MDP5001_342_I1_Channel_Active_Energy_1;
prgEM.stEL3446_IO_1.MDP5001_342_Input.MDP5001_342_I2_Channel_Overcurrent					:=	MDP5001_342_I2_Channel_Overcurrent_1;
prgEM.stEL3446_IO_1.MDP5001_342_Input.MDP5001_342_I2_Channel_Inaccurate_Current			:=	MDP5001_342_I2_Channel_Inaccurate_Current_1;
prgEM.stEL3446_IO_1.MDP5001_342_Input.MDP5001_342_I2_Channel_Current_Guard_Warning		:=	MDP5001_342_I2_Channel_Current_Guard_Warning_1;
prgEM.stEL3446_IO_1.MDP5001_342_Input.MDP5001_342_I2_Channel_Current_Guard_Error			:=	MDP5001_342_I2_Channel_Current_Guard_Error_1;
prgEM.stEL3446_IO_1.MDP5001_342_Input.MDP5001_342_I2_Channel_Apparent_Power_Guard_Warning	:=	MDP5001_342_I2_Channel_Apparent_Power_Guard_Warning_1;
prgEM.stEL3446_IO_1.MDP5001_342_Input.MDP5001_342_I2_Channel_Apparent_Power_Guard_Error	:=	MDP5001_342_I2_Channel_Apparent_Power_Guard_Error_1;
prgEM.stEL3446_IO_1.MDP5001_342_Input.MDP5001_342_I2_Channel_Active_Power_Guard_Warning	:=	MDP5001_342_I2_Channel_Active_Power_Guard_Warning_1;
prgEM.stEL3446_IO_1.MDP5001_342_Input.MDP5001_342_I2_Channel_Active_Power_Guard_Error		:=	MDP5001_342_I2_Channel_Active_Power_Guard_Error_1;
prgEM.stEL3446_IO_1.MDP5001_342_Input.MDP5001_342_I2_Channel_Reactive_Power_Guard_Warning	:=	MDP5001_342_I2_Channel_Reactive_Power_Guard_Warning_1;
prgEM.stEL3446_IO_1.MDP5001_342_Input.MDP5001_342_I2_Channel_Reactive_Power_Guard_Error	:=	MDP5001_342_I2_Channel_Reactive_Power_Guard_Error_1;
prgEM.stEL3446_IO_1.MDP5001_342_Input.MDP5001_342_I2_Channel_DPM_Inaccurate				:=	MDP5001_342_I2_Channel_DPM_Inaccurate_1;
prgEM.stEL3446_IO_1.MDP5001_342_Input.MDP5001_342_I2_Channel_DPM_Timeout					:=	MDP5001_342_I2_Channel_DPM_Timeout_1;
prgEM.stEL3446_IO_1.MDP5001_342_Input.MDP5001_342_I2_Channel_TxPDO_Toggle					:=	MDP5001_342_I2_Channel_TxPDO_Toggle_1;
prgEM.stEL3446_IO_1.MDP5001_342_Input.MDP5001_342_I2_Channel_Current						:=	MDP5001_342_I2_Channel_Current_1;
prgEM.stEL3446_IO_1.MDP5001_342_Input.MDP5001_342_I2_Channel_Active_Power					:=	MDP5001_342_I2_Channel_Active_Power_1;
prgEM.stEL3446_IO_1.MDP5001_342_Input.MDP5001_342_I2_Channel_Apparent_Power				:=	MDP5001_342_I2_Channel_Apparent_Power_1;
prgEM.stEL3446_IO_1.MDP5001_342_Input.MDP5001_342_I2_Channel_Reactive_Power_Fundamental	:=	MDP5001_342_I2_Channel_Reactive_Power_Fundamental_1;
prgEM.stEL3446_IO_1.MDP5001_342_Input.MDP5001_342_I2_Channel_Active_Energy				:=	MDP5001_342_I2_Channel_Active_Energy_1;
prgEM.stEL3446_IO_1.MDP5001_342_Input.MDP5001_342_I3_Channel_Overcurrent					:=	MDP5001_342_I3_Channel_Overcurrent_1;
prgEM.stEL3446_IO_1.MDP5001_342_Input.MDP5001_342_I3_Channel_Inaccurate_Current			:=	MDP5001_342_I3_Channel_Inaccurate_Current_1;
prgEM.stEL3446_IO_1.MDP5001_342_Input.MDP5001_342_I3_Channel_Current_Guard_Warning		:=	MDP5001_342_I3_Channel_Current_Guard_Warning_1;
prgEM.stEL3446_IO_1.MDP5001_342_Input.MDP5001_342_I3_Channel_Current_Guard_Error			:=	MDP5001_342_I3_Channel_Current_Guard_Error_1;
prgEM.stEL3446_IO_1.MDP5001_342_Input.MDP5001_342_I3_Channel_Apparent_Power_Guard_Warning	:=	MDP5001_342_I3_Channel_Apparent_Power_Guard_Warning_1;
prgEM.stEL3446_IO_1.MDP5001_342_Input.MDP5001_342_I3_Channel_Apparent_Power_Guard_Error	:=	MDP5001_342_I3_Channel_Apparent_Power_Guard_Error_1;
prgEM.stEL3446_IO_1.MDP5001_342_Input.MDP5001_342_I3_Channel_Active_Power_Guard_Warning	:=	MDP5001_342_I3_Channel_Active_Power_Guard_Warning_1;
prgEM.stEL3446_IO_1.MDP5001_342_Input.MDP5001_342_I3_Channel_Active_Power_Guard_Error		:=	MDP5001_342_I3_Channel_Active_Power_Guard_Error_1;
prgEM.stEL3446_IO_1.MDP5001_342_Input.MDP5001_342_I3_Channel_Reactive_Power_Guard_Warning	:=	MDP5001_342_I3_Channel_Reactive_Power_Guard_Warning_1;
prgEM.stEL3446_IO_1.MDP5001_342_Input.MDP5001_342_I3_Channel_Reactive_Power_Guard_Error	:=	MDP5001_342_I3_Channel_Reactive_Power_Guard_Error_1;
prgEM.stEL3446_IO_1.MDP5001_342_Input.MDP5001_342_I3_Channel_DPM_Inaccurate				:=	MDP5001_342_I3_Channel_DPM_Inaccurate_1;
prgEM.stEL3446_IO_1.MDP5001_342_Input.MDP5001_342_I3_Channel_DPM_Timeout					:=	MDP5001_342_I3_Channel_DPM_Timeout_1;
prgEM.stEL3446_IO_1.MDP5001_342_Input.MDP5001_342_I3_Channel_TxPDO_Toggle					:=	MDP5001_342_I3_Channel_TxPDO_Toggle_1;
prgEM.stEL3446_IO_1.MDP5001_342_Input.MDP5001_342_I3_Channel_Current						:=	MDP5001_342_I3_Channel_Current_1;
prgEM.stEL3446_IO_1.MDP5001_342_Input.MDP5001_342_I3_Channel_Active_Power					:=	MDP5001_342_I3_Channel_Active_Power_1;
prgEM.stEL3446_IO_1.MDP5001_342_Input.MDP5001_342_I3_Channel_Apparent_Power				:=	MDP5001_342_I3_Channel_Apparent_Power_1;
prgEM.stEL3446_IO_1.MDP5001_342_Input.MDP5001_342_I3_Channel_Reactive_Power_Fundamental	:=	MDP5001_342_I3_Channel_Reactive_Power_Fundamental_1;
prgEM.stEL3446_IO_1.MDP5001_342_Input.MDP5001_342_I3_Channel_Active_Energy				:=	MDP5001_342_I3_Channel_Active_Energy_1;
prgEM.stEL3446_IO_1.MDP5001_342_Input.MDP5001_342_I4_Channel_Overcurrent					:=	MDP5001_342_I4_Channel_Overcurrent_1;
prgEM.stEL3446_IO_1.MDP5001_342_Input.MDP5001_342_I4_Channel_Inaccurate_Current			:=	MDP5001_342_I4_Channel_Inaccurate_Current_1;
prgEM.stEL3446_IO_1.MDP5001_342_Input.MDP5001_342_I4_Channel_Current_Guard_Warning		:=	MDP5001_342_I4_Channel_Current_Guard_Warning_1;
prgEM.stEL3446_IO_1.MDP5001_342_Input.MDP5001_342_I4_Channel_Current_Guard_Error			:=	MDP5001_342_I4_Channel_Current_Guard_Error_1;
prgEM.stEL3446_IO_1.MDP5001_342_Input.MDP5001_342_I4_Channel_Apparent_Power_Guard_Warning	:=	MDP5001_342_I4_Channel_Apparent_Power_Guard_Warning_1;
prgEM.stEL3446_IO_1.MDP5001_342_Input.MDP5001_342_I4_Channel_Apparent_Power_Guard_Error	:=	MDP5001_342_I4_Channel_Apparent_Power_Guard_Error_1;
prgEM.stEL3446_IO_1.MDP5001_342_Input.MDP5001_342_I4_Channel_Active_Power_Guard_Warning	:=	MDP5001_342_I4_Channel_Active_Power_Guard_Warning_1;
prgEM.stEL3446_IO_1.MDP5001_342_Input.MDP5001_342_I4_Channel_Active_Power_Guard_Error		:=	MDP5001_342_I4_Channel_Active_Power_Guard_Error_1;
prgEM.stEL3446_IO_1.MDP5001_342_Input.MDP5001_342_I4_Channel_Reactive_Power_Guard_Warning	:=	MDP5001_342_I4_Channel_Reactive_Power_Guard_Warning_1;
prgEM.stEL3446_IO_1.MDP5001_342_Input.MDP5001_342_I4_Channel_Reactive_Power_Guard_Error	:=	MDP5001_342_I4_Channel_Reactive_Power_Guard_Error_1;
prgEM.stEL3446_IO_1.MDP5001_342_Input.MDP5001_342_I4_Channel_DPM_Inaccurate				:=	MDP5001_342_I4_Channel_DPM_Inaccurate_1;
prgEM.stEL3446_IO_1.MDP5001_342_Input.MDP5001_342_I4_Channel_DPM_Timeout					:=	MDP5001_342_I4_Channel_DPM_Timeout_1;
prgEM.stEL3446_IO_1.MDP5001_342_Input.MDP5001_342_I4_Channel_TxPDO_Toggle					:=	MDP5001_342_I4_Channel_TxPDO_Toggle_1;
prgEM.stEL3446_IO_1.MDP5001_342_Input.MDP5001_342_I4_Channel_Current						:=	MDP5001_342_I4_Channel_Current_1;
prgEM.stEL3446_IO_1.MDP5001_342_Input.MDP5001_342_I4_Channel_Active_Power					:=	MDP5001_342_I4_Channel_Active_Power_1;
prgEM.stEL3446_IO_1.MDP5001_342_Input.MDP5001_342_I4_Channel_Apparent_Power				:=	MDP5001_342_I4_Channel_Apparent_Power_1;
prgEM.stEL3446_IO_1.MDP5001_342_Input.MDP5001_342_I4_Channel_Reactive_Power_Fundamental	:=	MDP5001_342_I4_Channel_Reactive_Power_Fundamental_1;
prgEM.stEL3446_IO_1.MDP5001_342_Input.MDP5001_342_I4_Channel_Active_Energy				:=	MDP5001_342_I4_Channel_Active_Energy_1;
prgEM.stEL3446_IO_1.MDP5001_342_Input.MDP5001_342_I5_Channel_Overcurrent					:=	MDP5001_342_I5_Channel_Overcurrent_1;
prgEM.stEL3446_IO_1.MDP5001_342_Input.MDP5001_342_I5_Channel_Inaccurate_Current			:=	MDP5001_342_I5_Channel_Inaccurate_Current_1;
prgEM.stEL3446_IO_1.MDP5001_342_Input.MDP5001_342_I5_Channel_Current_Guard_Warning		:=	MDP5001_342_I5_Channel_Current_Guard_Warning_1;
prgEM.stEL3446_IO_1.MDP5001_342_Input.MDP5001_342_I5_Channel_Current_Guard_Error			:=	MDP5001_342_I5_Channel_Current_Guard_Error_1;
prgEM.stEL3446_IO_1.MDP5001_342_Input.MDP5001_342_I5_Channel_Apparent_Power_Guard_Warning	:=	MDP5001_342_I5_Channel_Apparent_Power_Guard_Warning_1;
prgEM.stEL3446_IO_1.MDP5001_342_Input.MDP5001_342_I5_Channel_Apparent_Power_Guard_Error	:=	MDP5001_342_I5_Channel_Apparent_Power_Guard_Error_1;
prgEM.stEL3446_IO_1.MDP5001_342_Input.MDP5001_342_I5_Channel_Active_Power_Guard_Warning	:=	MDP5001_342_I5_Channel_Active_Power_Guard_Warning_1;
prgEM.stEL3446_IO_1.MDP5001_342_Input.MDP5001_342_I5_Channel_Active_Power_Guard_Error		:=	MDP5001_342_I5_Channel_Active_Power_Guard_Error_1;
prgEM.stEL3446_IO_1.MDP5001_342_Input.MDP5001_342_I5_Channel_Reactive_Power_Guard_Warning	:=	MDP5001_342_I5_Channel_Reactive_Power_Guard_Warning_1;
prgEM.stEL3446_IO_1.MDP5001_342_Input.MDP5001_342_I5_Channel_Reactive_Power_Guard_Error	:=	MDP5001_342_I5_Channel_Reactive_Power_Guard_Error_1;
prgEM.stEL3446_IO_1.MDP5001_342_Input.MDP5001_342_I5_Channel_DPM_Inaccurate				:=	MDP5001_342_I5_Channel_DPM_Inaccurate_1;
prgEM.stEL3446_IO_1.MDP5001_342_Input.MDP5001_342_I5_Channel_DPM_Timeout					:=	MDP5001_342_I5_Channel_DPM_Timeout_1;
prgEM.stEL3446_IO_1.MDP5001_342_Input.MDP5001_342_I5_Channel_TxPDO_Toggle					:=	MDP5001_342_I5_Channel_TxPDO_Toggle_1;
prgEM.stEL3446_IO_1.MDP5001_342_Input.MDP5001_342_I5_Channel_Current						:=	MDP5001_342_I5_Channel_Current_1;
prgEM.stEL3446_IO_1.MDP5001_342_Input.MDP5001_342_I5_Channel_Active_Power					:=	MDP5001_342_I5_Channel_Active_Power_1;
prgEM.stEL3446_IO_1.MDP5001_342_Input.MDP5001_342_I5_Channel_Apparent_Power				:=	MDP5001_342_I5_Channel_Apparent_Power_1;
prgEM.stEL3446_IO_1.MDP5001_342_Input.MDP5001_342_I5_Channel_Reactive_Power_Fundamental	:=	MDP5001_342_I5_Channel_Reactive_Power_Fundamental_1;
prgEM.stEL3446_IO_1.MDP5001_342_Input.MDP5001_342_I5_Channel_Active_Energy				:=	MDP5001_342_I5_Channel_Active_Energy_1;
prgEM.stEL3446_IO_1.MDP5001_342_Input.MDP5001_342_I6_Channel_Overcurrent					:=	MDP5001_342_I6_Channel_Overcurrent_1;
prgEM.stEL3446_IO_1.MDP5001_342_Input.MDP5001_342_I6_Channel_Inaccurate_Current			:=	MDP5001_342_I6_Channel_Inaccurate_Current_1;
prgEM.stEL3446_IO_1.MDP5001_342_Input.MDP5001_342_I6_Channel_Current_Guard_Warning		:=	MDP5001_342_I6_Channel_Current_Guard_Warning_1;
prgEM.stEL3446_IO_1.MDP5001_342_Input.MDP5001_342_I6_Channel_Current_Guard_Error			:=	MDP5001_342_I6_Channel_Current_Guard_Error_1;
prgEM.stEL3446_IO_1.MDP5001_342_Input.MDP5001_342_I6_Channel_Apparent_Power_Guard_Warning	:=	MDP5001_342_I6_Channel_Apparent_Power_Guard_Warning_1;
prgEM.stEL3446_IO_1.MDP5001_342_Input.MDP5001_342_I6_Channel_Apparent_Power_Guard_Error	:=	MDP5001_342_I6_Channel_Apparent_Power_Guard_Error_1;
prgEM.stEL3446_IO_1.MDP5001_342_Input.MDP5001_342_I6_Channel_Active_Power_Guard_Warning	:=	MDP5001_342_I6_Channel_Active_Power_Guard_Warning_1;
prgEM.stEL3446_IO_1.MDP5001_342_Input.MDP5001_342_I6_Channel_Active_Power_Guard_Error		:=	MDP5001_342_I6_Channel_Active_Power_Guard_Error_1;
prgEM.stEL3446_IO_1.MDP5001_342_Input.MDP5001_342_I6_Channel_Reactive_Power_Guard_Warning	:=	MDP5001_342_I6_Channel_Reactive_Power_Guard_Warning_1;
prgEM.stEL3446_IO_1.MDP5001_342_Input.MDP5001_342_I6_Channel_Reactive_Power_Guard_Error	:=	MDP5001_342_I6_Channel_Reactive_Power_Guard_Error_1;
prgEM.stEL3446_IO_1.MDP5001_342_Input.MDP5001_342_I6_Channel_DPM_Inaccurate				:=	MDP5001_342_I6_Channel_DPM_Inaccurate_1;
prgEM.stEL3446_IO_1.MDP5001_342_Input.MDP5001_342_I6_Channel_DPM_Timeout					:=	MDP5001_342_I6_Channel_DPM_Timeout_1;
prgEM.stEL3446_IO_1.MDP5001_342_Input.MDP5001_342_I6_Channel_TxPDO_Toggle					:=	MDP5001_342_I6_Channel_TxPDO_Toggle_1;
prgEM.stEL3446_IO_1.MDP5001_342_Input.MDP5001_342_I6_Channel_Current						:=	MDP5001_342_I6_Channel_Current_1;
prgEM.stEL3446_IO_1.MDP5001_342_Input.MDP5001_342_I6_Channel_Active_Power					:=	MDP5001_342_I6_Channel_Active_Power_1;
prgEM.stEL3446_IO_1.MDP5001_342_Input.MDP5001_342_I6_Channel_Apparent_Power				:=	MDP5001_342_I6_Channel_Apparent_Power_1;
prgEM.stEL3446_IO_1.MDP5001_342_Input.MDP5001_342_I6_Channel_Reactive_Power_Fundamental	:=	MDP5001_342_I6_Channel_Reactive_Power_Fundamental_1;
prgEM.stEL3446_IO_1.MDP5001_342_Input.MDP5001_342_I6_Channel_Active_Energy				:=	MDP5001_342_I6_Channel_Active_Energy_1;
prgEM.stEL3446_IO_1.MDP5001_342_Input.MDP5001_342_DPM_Variant_Value_In_TxPDO_Toggle		:=	MDP5001_342_DPM_Variant_Value_In_TxPDO_Toggle_1;
prgEM.stEL3446_IO_1.MDP5001_342_Input.MDP5001_342_DPM_Variant_Value_In_Index_1_REAL		:=	MDP5001_342_DPM_Variant_Value_In_Index_1_REAL_1;
prgEM.stEL3446_IO_1.MDP5001_342_Input.MDP5001_342_DPM_Variant_Value_In_Value_1_REAL		:=	MDP5001_342_DPM_Variant_Value_In_Value_1_REAL_1;
prgEM.stEL3446_IO_1.MDP5001_342_Input.MDP5001_342_DPM_Variant_Value_In_Index_2_REAL		:=	MDP5001_342_DPM_Variant_Value_In_Index_2_REAL_1;
prgEM.stEL3446_IO_1.MDP5001_342_Input.MDP5001_342_DPM_Variant_Value_In_Value_2_REAL		:=	MDP5001_342_DPM_Variant_Value_In_Value_2_REAL_1;
prgEM.stEL3446_IO_1.MDP5001_342_Input.MDP5001_342_DPM_Variant_Value_In_Index_3_REAL		:=	MDP5001_342_DPM_Variant_Value_In_Index_3_REAL_1;
prgEM.stEL3446_IO_1.MDP5001_342_Input.MDP5001_342_DPM_Variant_Value_In_Value_3_REAL		:=	MDP5001_342_DPM_Variant_Value_In_Value_3_REAL_1;
prgEM.stEL3446_IO_1.MDP5001_342_Input.MDP5001_342_DPM_Variant_Value_In_Index_4_ULINT		:=	MDP5001_342_DPM_Variant_Value_In_Index_4_ULINT_1;
prgEM.stEL3446_IO_1.MDP5001_342_Input.MDP5001_342_DPM_Variant_Value_In_Value_4_ULINT		:=	MDP5001_342_DPM_Variant_Value_In_Value_4_ULINT_1;

MDP5001_342_DPM_Variant_Value_Out_Index_1_REAL_1	:= 		prgEM.stEL3446_IO_1.MDP5001_342_Output.MDP5001_342_DPM_Variant_Value_Out_Index_1_REAL	;
MDP5001_342_DPM_Variant_Value_Out_Index_2_REAL_1	:= 		prgEM.stEL3446_IO_1.MDP5001_342_Output.MDP5001_342_DPM_Variant_Value_Out_Index_2_REAL	;	
MDP5001_342_DPM_Variant_Value_Out_Index_3_REAL_1	:= 		prgEM.stEL3446_IO_1.MDP5001_342_Output.MDP5001_342_DPM_Variant_Value_Out_Index_3_REAL	;
MDP5001_342_DPM_Variant_Value_Out_Index_4_ULINT_1	:= 		prgEM.stEL3446_IO_1.MDP5001_342_Output.MDP5001_342_DPM_Variant_Value_Out_Index_4_ULINT	;
MDP5001_342_DPM_Data_Data_1_1						:= 		prgEM.stEL3446_IO_1.MDP5001_342_Output.MDP5001_342_DPM_Data_Data_1	;
MDP5001_342_DPM_Data_Data_2_1						:= 		prgEM.stEL3446_IO_1.MDP5001_342_Output.MDP5001_342_DPM_Data_Data_2	;
MDP5001_342_DPM_Data_Data_3_1						:= 		prgEM.stEL3446_IO_1.MDP5001_342_Output.MDP5001_342_DPM_Data_Data_3	;
MDP5001_342_DPM_Data_Data_4_1						:= 		prgEM.stEL3446_IO_1.MDP5001_342_Output.MDP5001_342_DPM_Data_Data_4	;
MDP5001_342_DPM_Data_Data_5_1						:= 		prgEM.stEL3446_IO_1.MDP5001_342_Output.MDP5001_342_DPM_Data_Data_5	;
MDP5001_342_DPM_Data_Data_6_1						:= 		prgEM.stEL3446_IO_1.MDP5001_342_Output.MDP5001_342_DPM_Data_Data_6	;
MDP5001_342_DPM_Data_Data_7_1						:= 		prgEM.stEL3446_IO_1.MDP5001_342_Output.MDP5001_342_DPM_Data_Data_7	;
MDP5001_342_DPM_Data_Data_8_1						:= 		prgEM.stEL3446_IO_1.MDP5001_342_Output.MDP5001_342_DPM_Data_Data_8	;
MDP5001_342_DPM_Data_Data_9_1						:= 		prgEM.stEL3446_IO_1.MDP5001_342_Output.MDP5001_342_DPM_Data_Data_9	;
MDP5001_342_DPM_Data_Data_10_1						:= 		prgEM.stEL3446_IO_1.MDP5001_342_Output.MDP5001_342_DPM_Data_Data_10	;
MDP5001_342_DPM_Data_Data_11_1						:= 		prgEM.stEL3446_IO_1.MDP5001_342_Output.MDP5001_342_DPM_Data_Data_11	;
MDP5001_342_DPM_Data_Data_12_1						:= 		prgEM.stEL3446_IO_1.MDP5001_342_Output.MDP5001_342_DPM_Data_Data_12	;
MDP5001_342_DPM_Data_Data_13_1						:= 		prgEM.stEL3446_IO_1.MDP5001_342_Output.MDP5001_342_DPM_Data_Data_13	;
MDP5001_342_DPM_Data_Data_14_1						:= 		prgEM.stEL3446_IO_1.MDP5001_342_Output.MDP5001_342_DPM_Data_Data_14	;
MDP5001_342_DPM_Data_Data_15_1						:= 		prgEM.stEL3446_IO_1.MDP5001_342_Output.MDP5001_342_DPM_Data_Data_15	;
MDP5001_342_DPM_Data_Data_16_1						:= 		prgEM.stEL3446_IO_1.MDP5001_342_Output.MDP5001_342_DPM_Data_Data_16	;
MDP5001_342_DPM_Data_Data_17_1						:= 		prgEM.stEL3446_IO_1.MDP5001_342_Output.MDP5001_342_DPM_Data_Data_17	;
MDP5001_342_DPM_Data_Data_18_1						:= 		prgEM.stEL3446_IO_1.MDP5001_342_Output.MDP5001_342_DPM_Data_Data_18	;
MDP5001_342_DPM_Data_Data_19_1						:= 		prgEM.stEL3446_IO_1.MDP5001_342_Output.MDP5001_342_DPM_Data_Data_19	;
MDP5001_342_DPM_Data_Data_20_1						:= 		prgEM.stEL3446_IO_1.MDP5001_342_Output.MDP5001_342_DPM_Data_Data_20	;




